LIN {X 0,Y 385.59,Z 292.202,A -85,B 0,C 180,E1 18203.536,E2 18203.536} C_VEL
LIN {X 0,Y 385.578,Z 292.169,A -85,B 0,C 180,E1 18199.701,E2 18199.701} C_VEL
LIN {X 0,Y 385.573,Z 292.168,A -85,B 0,C 180,E1 18195.8,E2 18195.8} C_VEL
LIN {X 0,Y 385.58,Z 292.204,A -85,B 0,C 180,E1 18191.821,E2 18191.821} C_VEL
LIN {X 0,Y 385.579,Z 292.173,A -85,B 0,C 180,E1 18187.75,E2 18187.75} C_VEL
LIN {X 0,Y 385.579,Z 292.168,A -85,B 0,C 180,E1 18183.717,E2 18183.717} C_VEL
LIN {X 0,Y 385.585,Z 292.205,A -85,B 0,C 180,E1 18179.703,E2 18179.703} C_VEL
LIN {X 0,Y 385.583,Z 292.167,A -85,B 0,C 180,E1 18175.687,E2 18175.687} C_VEL
LIN {X 0,Y 385.585,Z 292.173,A -85,B 0,C 180,E1 18171.65,E2 18171.65} C_VEL
LIN {X 0,Y 385.589,Z 292.205,A -85,B 0,C 180,E1 18167.571,E2 18167.571} C_VEL
LIN {X 0,Y 385.589,Z 292.169,A -85,B 0,C 180,E1 18163.582,E2 18163.582} C_VEL
LIN {X 0,Y 385.597,Z 292.203,A -85,B 0,C 180,E1 18159.668,E2 18159.668} C_VEL
LIN {X 0,Y 385.607,Z 292.202,A -85,B 0,C 180,E1 18155.815,E2 18155.815} C_VEL
LIN {X 0,Y 385.613,Z 292.203,A -85,B 0,C 180,E1 18151.831,E2 18151.831} C_VEL
LIN {X 0,Y 385.617,Z 292.201,A -85,B 0,C 180,E1 18147.891,E2 18147.891} C_VEL
LIN {X 0,Y 385.62,Z 292.2,A -85,B 0,C 180,E1 18143.944,E2 18143.944} C_VEL
LIN {X 0,Y 385.628,Z 292.199,A -85,B 0,C 180,E1 18139.894,E2 18139.894} C_VEL
LIN {X 0,Y 385.622,Z 292.201,A -85,B 0,C 180,E1 18135.775,E2 18135.775} C_VEL
LIN {X 0,Y 385.627,Z 292.203,A -85,B 0,C 180,E1 18131.692,E2 18131.692} C_VEL
LIN {X 0,Y 385.625,Z 292.202,A -85,B 0,C 180,E1 18127.726,E2 18127.726} C_VEL
LIN {X 0,Y 385.628,Z 292.234,A -85,B 0,C 180,E1 18123.666,E2 18123.666} C_VEL
LIN {X 0,Y 385.77,Z 293.033,A -85,B 0,C 180,E1 18121.396,E2 18121.396} C_VEL
LIN {X 0,Y 387.406,Z 296.314,A -85,B 0,C 180,E1 18118.016,E2 18118.016} C_VEL
LIN {X 0,Y 389.142,Z 297.888,A -85,B 0,C 180,E1 18114.759,E2 18114.759} C_VEL
LIN {X 0,Y 390.851,Z 298.757,A -85,B 0,C 180,E1 18111.3,E2 18111.3} C_VEL
LIN {X 0,Y 392.259,Z 299.662,A -85,B 0,C 180,E1 18107.964,E2 18107.964} C_VEL
LIN {X 0,Y 393.297,Z 301.626,A -85,B 0,C 180,E1 18104.727,E2 18104.727} C_VEL
LIN {X 0,Y 394.199,Z 303.074,A -85,B 0,C 180,E1 18101.262,E2 18101.262} C_VEL
LIN {X 0,Y 394.882,Z 303.844,A -85,B 0,C 180,E1 18097.712,E2 18097.712} C_VEL
LIN {X 0,Y 395.319,Z 304.24,A -85,B 0,C 180,E1 18094.206,E2 18094.206} C_VEL
LIN {X 0,Y 395.491,Z 304.381,A -85,B 0,C 180,E1 18090.724,E2 18090.724} C_VEL
LIN {X 0,Y 395.407,Z 304.311,A -85,B 0,C 180,E1 18087.101,E2 18087.101} C_VEL
LIN {X 0,Y 395.034,Z 303.985,A -85,B 0,C 180,E1 18083.46,E2 18083.46} C_VEL
LIN {X 0,Y 394.383,Z 303.295,A -85,B 0,C 180,E1 18079.778,E2 18079.778} C_VEL
LIN {X 0,Y 393.61,Z 302.209,A -85,B 0,C 180,E1 18076.485,E2 18076.485} C_VEL
LIN {X 0,Y 392.679,Z 300.302,A -85,B 0,C 180,E1 18073.126,E2 18073.126} C_VEL
LIN {X 0,Y 391.442,Z 298.996,A -85,B 0,C 180,E1 18069.985,E2 18069.985} C_VEL
LIN {X 0,Y 389.81,Z 298.272,A -85,B 0,C 180,E1 18066.574,E2 18066.574} C_VEL
LIN {X 0,Y 387.974,Z 296.947,A -85,B 0,C 180,E1 18063.085,E2 18063.085} C_VEL
LIN {X 0,Y 387.725,Z 296.681,A -85,B 0,C 180,E1 18062.634,E2 18062.634} C_VEL
LIN {X 0,Y 387.23,Z 297.203,A -85,B 0,C 180,E1 18061.86,E2 18061.86} C_VEL
LIN {X 0,Y 385.442,Z 301.535,A -85,B 0,C 180,E1 18059.944,E2 18059.944} C_VEL
LIN {X 0,Y 384.858,Z 301.636,A -85,B 0,C 180,E1 18059.176,E2 18059.176} C_VEL
LIN {X 0,Y 383.634,Z 300.068,A -85,B 0,C 180,E1 18057.174,E2 18057.174} C_VEL
LIN {X 0,Y 381.125,Z 298.816,A -85,B 0,C 180,E1 18053.638,E2 18053.638} C_VEL
LIN {X 0,Y 379.099,Z 296.853,A -85,B 0,C 180,E1 18050.842,E2 18050.842} C_VEL
LIN {X 0,Y 377.788,Z 293.814,A -85,B 0,C 180,E1 18048.373,E2 18048.373} C_VEL
LIN {X 0,Y 377.677,Z 293.211,A -85,B 0,C 180,E1 18046.501,E2 18046.501} C_VEL
LIN {X 0,Y 377.676,Z 293.192,A -85,B 0,C 180,E1 18042.388,E2 18042.388} C_VEL
LIN {X 0,Y 377.672,Z 293.193,A -85,B 0,C 180,E1 18038.407,E2 18038.407} C_VEL
LIN {X 0,Y 377.67,Z 293.192,A -85,B 0,C 180,E1 18034.312,E2 18034.312} C_VEL
LIN {X 0,Y 377.668,Z 293.193,A -85,B 0,C 180,E1 18030.34,E2 18030.34} C_VEL
LIN {X 0,Y 377.662,Z 293.192,A -85,B 0,C 180,E1 18026.409,E2 18026.409} C_VEL
LIN {X 0,Y 377.657,Z 293.194,A -85,B 0,C 180,E1 18022.411,E2 18022.411} C_VEL
LIN {X 0,Y 377.658,Z 293.194,A -85,B 0,C 180,E1 18018.364,E2 18018.364} C_VEL
LIN {X 0,Y 377.651,Z 293.162,A -85,B 0,C 180,E1 18014.254,E2 18014.254} C_VEL
LIN {X 0,Y 377.648,Z 293.151,A -85,B 0,C 180,E1 18010.218,E2 18010.218} C_VEL
LIN {X 0,Y 377.65,Z 293.194,A -85,B 0,C 180,E1 18006.232,E2 18006.232} C_VEL
LIN {X 0,Y 377.645,Z 293.16,A -85,B 0,C 180,E1 18002.124,E2 18002.124} C_VEL
LIN {X 0,Y 377.641,Z 293.155,A -85,B 0,C 180,E1 17998.179,E2 17998.179} C_VEL
LIN {X 0,Y 377.646,Z 293.194,A -85,B 0,C 180,E1 17994.073,E2 17994.073} C_VEL
LIN {X 0,Y 377.638,Z 293.157,A -85,B 0,C 180,E1 17990.031,E2 17990.031} C_VEL
LIN {X 0,Y 377.634,Z 293.159,A -85,B 0,C 180,E1 17986.058,E2 17986.058} C_VEL
LIN {X 0,Y 377.639,Z 293.195,A -85,B 0,C 180,E1 17981.954,E2 17981.954} C_VEL
LIN {X 0,Y 377.633,Z 293.172,A -85,B 0,C 180,E1 17977.916,E2 17977.916} C_VEL
LIN {X 0,Y 377.631,Z 293.159,A -85,B 0,C 180,E1 17973.838,E2 17973.838} C_VEL
LIN {X 0,Y 377.655,Z 293.299,A -85,B 0,C 180,E1 17970.237,E2 17970.237} C_VEL
LIN {X 0,Y 378.612,Z 296.099,A -85,B 0,C 180,E1 17969.269,E2 17969.269} C_VEL
LIN {X 0,Y 383.609,Z 302.624,A -85,B 0,C 180,E1 17967.79,E2 17967.79} C_VEL
LIN {X 0,Y 391.931,Z 314.43,A -85,B 0,C 180,E1 17965.549,E2 17965.549} C_VEL
LIN {X 0,Y 395.837,Z 319.96,A -85,B 0,C 180,E1 17964.571,E2 17964.571} C_VEL
LIN {X 0,Y 403.618,Z 331.65,A -85,B 0,C 180,E1 17962.722,E2 17962.722} C_VEL
LIN {X 0,Y 410.877,Z 343.12,A -85,B 0,C 180,E1 17961.109,E2 17961.109} C_VEL
LIN {X 0,Y 420.09,Z 358.902,A -85,B 0,C 180,E1 17959.184,E2 17959.184} C_VEL
LIN {X 0,Y 426.598,Z 371.081,A -85,B 0,C 180,E1 17957.891,E2 17957.891} C_VEL
LIN {X 0,Y 418.324,Z 587.742,A -85,B 0,C 180,E1 17953.875,E2 17953.875} C_VEL
LIN {X 0,Y 416.849,Z 613.236,A -85,B 0,C 180,E1 17953.319,E2 17953.319} C_VEL
LIN {X 0,Y 415.022,Z 632.082,A -85,B 0,C 180,E1 17952.735,E2 17952.735} C_VEL
LIN {X 0,Y 412.471,Z 653.444,A -85,B 0,C 180,E1 17951.852,E2 17951.852} C_VEL
LIN {X 0,Y 409.295,Z 674.289,A -85,B 0,C 180,E1 17950.71,E2 17950.71} C_VEL
LIN {X 0,Y 406.38,Z 691.177,A -85,B 0,C 180,E1 17949.585,E2 17949.585} C_VEL
LIN {X 0,Y 402.808,Z 710.1,A -85,B 0,C 180,E1 17948.084,E2 17948.084} C_VEL
LIN {X 0,Y 398.872,Z 728.796,A -85,B 0,C 180,E1 17946.268,E2 17946.268} C_VEL
LIN {X 0,Y 395.578,Z 743.764,A -85,B 0,C 180,E1 17944.571,E2 17944.571} C_VEL
LIN {X 0,Y 391.775,Z 760.597,A -85,B 0,C 180,E1 17942.355,E2 17942.355} C_VEL
LIN {X 0,Y 388.258,Z 775.729,A -85,B 0,C 180,E1 17939.972,E2 17939.972} C_VEL
LIN {X 0,Y 385.567,Z 787.594,A -85,B 0,C 180,E1 17937.825,E2 17937.825} C_VEL
LIN {X 0,Y 382.708,Z 800.935,A -85,B 0,C 180,E1 17935.039,E2 17935.039} C_VEL
LIN {X 0,Y 380.326,Z 812.676,A -85,B 0,C 180,E1 17932.082,E2 17932.082} C_VEL
LIN {X 0,Y 378.728,Z 821.683,A -85,B 0,C 180,E1 17929.429,E2 17929.429} C_VEL
LIN {X 0,Y 377.359,Z 830.966,A -85,B 0,C 180,E1 17926.153,E2 17926.153} C_VEL
LIN {X 0,Y 376.588,Z 837.631,A -85,B 0,C 180,E1 17923.199,E2 17923.199} C_VEL
LIN {X 0,Y 376.187,Z 842.608,A -85,B 0,C 180,E1 17920.451,E2 17920.451} C_VEL
LIN {X 0,Y 375.986,Z 846.946,A -85,B 0,C 180,E1 17917.291,E2 17917.291} C_VEL
LIN {X 0,Y 375.927,Z 849.714,A -85,B 0,C 180,E1 17913.965,E2 17913.965} C_VEL
LIN {X 0,Y 375.926,Z 850.752,A -85,B 0,C 180,E1 17911.372,E2 17911.372} C_VEL
LIN {X 0,Y 375.928,Z 850.78,A -85,B 0,C 180,E1 17908.781,E2 17908.781} C_VEL
LIN {X 0,Y 375.927,Z 849.797,A -85,B 0,C 180,E1 17906.188,E2 17906.188} C_VEL
LIN {X 0,Y 375.969,Z 847.379,A -85,B 0,C 180,E1 17903.127,E2 17903.127} C_VEL
LIN {X 0,Y 376.166,Z 842.922,A -85,B 0,C 180,E1 17899.742,E2 17899.742} C_VEL
LIN {X 0,Y 376.558,Z 837.942,A -85,B 0,C 180,E1 17896.957,E2 17896.957} C_VEL
LIN {X 0,Y 377.309,Z 831.337,A -85,B 0,C 180,E1 17894.003,E2 17894.003} C_VEL
LIN {X 0,Y 378.651,Z 822.182,A -85,B 0,C 180,E1 17890.727,E2 17890.727} C_VEL
LIN {X 0,Y 380.22,Z 813.244,A -85,B 0,C 180,E1 17888.074,E2 17888.074} C_VEL
LIN {X 0,Y 382.277,Z 802.862,A -85,B 0,C 180,E1 17885.427,E2 17885.427} C_VEL
LIN {X 0,Y 385.215,Z 789.2,A -85,B 0,C 180,E1 17882.484,E2 17882.484} C_VEL
LIN {X 0,Y 388.052,Z 776.624,A -85,B 0,C 180,E1 17880.18,E2 17880.18} C_VEL
LIN {X 0,Y 391.238,Z 762.786,A -85,B 0,C 180,E1 17877.976,E2 17877.976} C_VEL
LIN {X 0,Y 395.321,Z 744.936,A -85,B 0,C 180,E1 17875.57,E2 17875.57} C_VEL
LIN {X 0,Y 398.708,Z 729.554,A -85,B 0,C 180,E1 17873.812,E2 17873.812} C_VEL
LIN {X 0,Y 402.305,Z 712.451,A -85,B 0,C 180,E1 17872.131,E2 17872.131} C_VEL
LIN {X 0,Y 406.204,Z 692.165,A -85,B 0,C 180,E1 17870.486,E2 17870.486} C_VEL
LIN {X 0,Y 409.103,Z 675.423,A -85,B 0,C 180,E1 17869.359,E2 17869.359} C_VEL
LIN {X 0,Y 411.972,Z 656.79,A -85,B 0,C 180,E1 17868.319,E2 17868.319} C_VEL
LIN {X 0,Y 414.823,Z 634.055,A -85,B 0,C 180,E1 17867.336,E2 17867.336} C_VEL
LIN {X 0,Y 416.669,Z 615.37,A -85,B 0,C 180,E1 17866.74,E2 17866.74} C_VEL
LIN {X 0,Y 418.066,Z 594.306,A -85,B 0,C 180,E1 17866.25,E2 17866.25} C_VEL
LIN {X 0,Y 426.442,Z 375.04,A -85,B 0,C 180,E1 17862.183,E2 17862.183} C_VEL
LIN {X 0,Y 426.491,Z 370.624,A -85,B 0,C 180,E1 17862.082,E2 17862.082} C_VEL
LIN {X 0,Y 416.389,Z 352.336,A -85,B 0,C 180,E1 17860.056,E2 17860.056} C_VEL
LIN {X 0,Y 405.621,Z 334.64,A -85,B 0,C 180,E1 17857.73,E2 17857.73} C_VEL
LIN {X 0,Y 396.092,Z 320.326,A -85,B 0,C 180,E1 17855.492,E2 17855.492} C_VEL
LIN {X 0,Y 392.43,Z 315.132,A -85,B 0,C 180,E1 17854.579,E2 17854.579} C_VEL
LIN {X 0,Y 386.918,Z 307.383,A -85,B 0,C 180,E1 17853.131,E2 17853.131} C_VEL
LIN {X 0,Y 383.245,Z 302.265,A -85,B 0,C 180,E1 17852.111,E2 17852.111} C_VEL
LIN {X 0,Y 378.455,Z 295.814,A -85,B 0,C 180,E1 17850.657,E2 17850.657} C_VEL
LIN {X 0,Y 377.652,Z 293.269,A -85,B 0,C 180,E1 17849.729,E2 17849.729} C_VEL
LIN {X 0,Y 377.637,Z 293.156,A -85,B 0,C 180,E1 17845.735,E2 17845.735} C_VEL
LIN {X 0,Y 377.631,Z 293.166,A -85,B 0,C 180,E1 17841.921,E2 17841.921} C_VEL
LIN {X 0,Y 377.639,Z 293.192,A -85,B 0,C 180,E1 17837.886,E2 17837.886} C_VEL
LIN {X 0,Y 377.635,Z 293.159,A -85,B 0,C 180,E1 17833.786,E2 17833.786} C_VEL
LIN {X 0,Y 377.637,Z 293.153,A -85,B 0,C 180,E1 17829.756,E2 17829.756} C_VEL
LIN {X 0,Y 377.644,Z 293.195,A -85,B 0,C 180,E1 17825.774,E2 17825.774} C_VEL
LIN {X 0,Y 377.641,Z 293.158,A -85,B 0,C 180,E1 17821.669,E2 17821.669} C_VEL
LIN {X 0,Y 377.643,Z 293.157,A -85,B 0,C 180,E1 17817.724,E2 17817.724} C_VEL
LIN {X 0,Y 377.648,Z 293.194,A -85,B 0,C 180,E1 17813.616,E2 17813.616} C_VEL
LIN {X 0,Y 377.647,Z 293.155,A -85,B 0,C 180,E1 17809.474,E2 17809.474} C_VEL
LIN {X 0,Y 377.647,Z 293.157,A -85,B 0,C 180,E1 17805.432,E2 17805.432} C_VEL
LIN {X 0,Y 377.657,Z 293.194,A -85,B 0,C 180,E1 17801.316,E2 17801.316} C_VEL
LIN {X 0,Y 377.659,Z 293.193,A -85,B 0,C 180,E1 17797.261,E2 17797.261} C_VEL
LIN {X 0,Y 377.663,Z 293.192,A -85,B 0,C 180,E1 17793.148,E2 17793.148} C_VEL
LIN {X 0,Y 377.663,Z 293.19,A -85,B 0,C 180,E1 17789.066,E2 17789.066} C_VEL
LIN {X 0,Y 377.664,Z 293.191,A -85,B 0,C 180,E1 17785.12,E2 17785.12} C_VEL
LIN {X 0,Y 377.664,Z 293.19,A -85,B 0,C 180,E1 17781.109,E2 17781.109} C_VEL
LIN {X 0,Y 377.666,Z 293.189,A -85,B 0,C 180,E1 17777.125,E2 17777.125} C_VEL
LIN {X 0,Y 377.671,Z 293.229,A -85,B 0,C 180,E1 17773.056,E2 17773.056} C_VEL
LIN {X 0,Y 377.86,Z 294.198,A -85,B 0,C 180,E1 17771.213,E2 17771.213} C_VEL
LIN {X 0,Y 379.306,Z 297.127,A -85,B 0,C 180,E1 17768.855,E2 17768.855} C_VEL
LIN {X 0,Y 381.485,Z 299.049,A -85,B 0,C 180,E1 17765.916,E2 17765.916} C_VEL
LIN {X 0,Y 384.034,Z 300.4,A -85,B 0,C 180,E1 17762.257,E2 17762.257} C_VEL
LIN {X 0,Y 385.148,Z 302.283,A -85,B 0,C 180,E1 17760.326,E2 17760.326} C_VEL
LIN {X 0,Y 386.727,Z 304.625,A -85,B 0,C 180,E1 17757.4,E2 17757.4} C_VEL
LIN {X 0,Y 388.497,Z 306.031,A -85,B 0,C 180,E1 17754.155,E2 17754.155} C_VEL
LIN {X 0,Y 390.264,Z 306.859,A -85,B 0,C 180,E1 17750.548,E2 17750.548} C_VEL
LIN {X 0,Y 391.49,Z 307.922,A -85,B 0,C 180,E1 17747.386,E2 17747.386} C_VEL
LIN {X 0,Y 392.489,Z 309.904,A -85,B 0,C 180,E1 17744.005,E2 17744.005} C_VEL
LIN {X 0,Y 393.317,Z 311.132,A -85,B 0,C 180,E1 17740.694,E2 17740.694} C_VEL
LIN {X 0,Y 393.988,Z 311.849,A -85,B 0,C 180,E1 17737.29,E2 17737.29} C_VEL
LIN {X 0,Y 394.418,Z 312.249,A -85,B 0,C 180,E1 17733.633,E2 17733.633} C_VEL
LIN {X 0,Y 394.573,Z 312.362,A -85,B 0,C 180,E1 17730,E2 17730} C_VEL
LIN {X 0,Y 394.419,Z 312.25,A -85,B 0,C 180,E1 17726.367,E2 17726.367} C_VEL
LIN {X 0,Y 393.988,Z 311.849,A -85,B 0,C 180,E1 17722.71,E2 17722.71} C_VEL
LIN {X 0,Y 393.294,Z 311.102,A -85,B 0,C 180,E1 17719.157,E2 17719.157} C_VEL
LIN {X 0,Y 392.451,Z 309.82,A -85,B 0,C 180,E1 17715.843,E2 17715.843} C_VEL
LIN {X 0,Y 391.374,Z 307.737,A -85,B 0,C 180,E1 17712.302,E2 17712.302} C_VEL
LIN {X 0,Y 390.013,Z 306.761,A -85,B 0,C 180,E1 17708.967,E2 17708.967} C_VEL
LIN {X 0,Y 388.245,Z 305.89,A -85,B 0,C 180,E1 17705.38,E2 17705.38} C_VEL
LIN {X 0,Y 386.47,Z 304.328,A -85,B 0,C 180,E1 17702.078,E2 17702.078} C_VEL
LIN {X 0,Y 384.882,Z 301.692,A -85,B 0,C 180,E1 17699.219,E2 17699.219} C_VEL
LIN {X 0,Y 384.858,Z 301.636,A -85,B 0,C 180,E1 17699.176,E2 17699.176} C_VEL
LIN {X 0,Y 384.246,Z 301.381,A -85,B 0,C 180,E1 17698.194,E2 17698.194} C_VEL
LIN {X 0,Y 382.956,Z 303.453,A -85,B 0,C 180,E1 17696.736,E2 17696.736} C_VEL
LIN {X 0,Y 381.184,Z 306.655,A -85,B 0,C 180,E1 17694.862,E2 17694.862} C_VEL
LIN {X 0,Y 380.383,Z 306.928,A -85,B 0,C 180,E1 17693.941,E2 17693.941} C_VEL
LIN {X 0,Y 378.223,Z 305,A -85,B 0,C 180,E1 17691.006,E2 17691.006} C_VEL
LIN {X 0,Y 376.839,Z 302.509,A -85,B 0,C 180,E1 17689.011,E2 17689.011} C_VEL
LIN {X 0,Y 375.463,Z 300.938,A -85,B 0,C 180,E1 17687.231,E2 17687.231} C_VEL
LIN {X 0,Y 372.507,Z 299.283,A -85,B 0,C 180,E1 17683.779,E2 17683.779} C_VEL
LIN {X 0,Y 370.823,Z 297.29,A -85,B 0,C 180,E1 17681.758,E2 17681.758} C_VEL
LIN {X 0,Y 369.822,Z 294.627,A -85,B 0,C 180,E1 17679.843,E2 17679.843} C_VEL
LIN {X 0,Y 369.729,Z 294.177,A -85,B 0,C 180,E1 17677.085,E2 17677.085} C_VEL
LIN {X 0,Y 369.725,Z 294.179,A -85,B 0,C 180,E1 17672.927,E2 17672.927} C_VEL
LIN {X 0,Y 369.721,Z 294.18,A -85,B 0,C 180,E1 17668.775,E2 17668.775} C_VEL
LIN {X 0,Y 369.72,Z 294.183,A -85,B 0,C 180,E1 17664.612,E2 17664.612} C_VEL
LIN {X 0,Y 369.718,Z 294.182,A -85,B 0,C 180,E1 17660.583,E2 17660.583} C_VEL
LIN {X 0,Y 369.708,Z 294.145,A -85,B 0,C 180,E1 17656.497,E2 17656.497} C_VEL
LIN {X 0,Y 369.712,Z 294.182,A -85,B 0,C 180,E1 17652.336,E2 17652.336} C_VEL
LIN {X 0,Y 369.71,Z 294.149,A -85,B 0,C 180,E1 17648.192,E2 17648.192} C_VEL
LIN {X 0,Y 369.706,Z 294.139,A -85,B 0,C 180,E1 17644.187,E2 17644.187} C_VEL
LIN {X 0,Y 369.708,Z 294.183,A -85,B 0,C 180,E1 17640.155,E2 17640.155} C_VEL
LIN {X 0,Y 369.701,Z 294.144,A -85,B 0,C 180,E1 17636.123,E2 17636.123} C_VEL
LIN {X 0,Y 369.7,Z 294.145,A -85,B 0,C 180,E1 17632.072,E2 17632.072} C_VEL
LIN {X 0,Y 369.704,Z 294.184,A -85,B 0,C 180,E1 17627.981,E2 17627.981} C_VEL
LIN {X 0,Y 369.697,Z 294.148,A -85,B 0,C 180,E1 17623.987,E2 17623.987} C_VEL
LIN {X 0,Y 369.694,Z 294.144,A -85,B 0,C 180,E1 17619.911,E2 17619.911} C_VEL
LIN {X 0,Y 369.695,Z 294.165,A -85,B 0,C 180,E1 17615.897,E2 17615.897} C_VEL
LIN {X 0,Y 369.719,Z 294.354,A -85,B 0,C 180,E1 17612.017,E2 17612.017} C_VEL
LIN {X 0,Y 370.014,Z 295.612,A -85,B 0,C 180,E1 17611.58,E2 17611.58} C_VEL
LIN {X 0,Y 371.953,Z 298.759,A -85,B 0,C 180,E1 17610.886,E2 17610.886} C_VEL
LIN {X 0,Y 374.407,Z 301.301,A -85,B 0,C 180,E1 17610.129,E2 17610.129} C_VEL
LIN {X 0,Y 381.676,Z 310.922,A -85,B 0,C 180,E1 17607.962,E2 17607.962} C_VEL
LIN {X 0,Y 388.476,Z 320.636,A -85,B 0,C 180,E1 17606.092,E2 17606.092} C_VEL
LIN {X 0,Y 395.873,Z 331.318,A -85,B 0,C 180,E1 17604.218,E2 17604.218} C_VEL
LIN {X 0,Y 404.594,Z 345.229,A -85,B 0,C 180,E1 17602.158,E2 17602.158} C_VEL
LIN {X 0,Y 413.34,Z 359.909,A -85,B 0,C 180,E1 17600.244,E2 17600.244} C_VEL
LIN {X 0,Y 421.1,Z 374.389,A -85,B 0,C 180,E1 17598.635,E2 17598.635} C_VEL
LIN {X 0,Y 412.376,Z 592.617,A -85,B 0,C 180,E1 17594.552,E2 17594.552} C_VEL
LIN {X 0,Y 410.888,Z 614.663,A -85,B 0,C 180,E1 17594.041,E2 17594.041} C_VEL
LIN {X 0,Y 408.974,Z 633.378,A -85,B 0,C 180,E1 17593.445,E2 17593.445} C_VEL
LIN {X 0,Y 406.172,Z 655.22,A -85,B 0,C 180,E1 17592.509,E2 17592.509} C_VEL
LIN {X 0,Y 403.179,Z 674.037,A -85,B 0,C 180,E1 17591.462,E2 17591.462} C_VEL
LIN {X 0,Y 400.137,Z 690.924,A -85,B 0,C 180,E1 17590.328,E2 17590.328} C_VEL
LIN {X 0,Y 396.328,Z 710.208,A -85,B 0,C 180,E1 17588.781,E2 17588.781} C_VEL
LIN {X 0,Y 392.272,Z 728.541,A -85,B 0,C 180,E1 17586.979,E2 17586.979} C_VEL
LIN {X 0,Y 388.813,Z 743.507,A -85,B 0,C 180,E1 17585.261,E2 17585.261} C_VEL
LIN {X 0,Y 384.767,Z 760.538,A -85,B 0,C 180,E1 17582.983,E2 17582.983} C_VEL
LIN {X 0,Y 381.096,Z 775.471,A -85,B 0,C 180,E1 17580.595,E2 17580.595} C_VEL
LIN {X 0,Y 378.108,Z 787.963,A -85,B 0,C 180,E1 17578.288,E2 17578.288} C_VEL
LIN {X 0,Y 374.904,Z 801.963,A -85,B 0,C 180,E1 17575.259,E2 17575.259} C_VEL
LIN {X 0,Y 372.668,Z 812.419,A -85,B 0,C 180,E1 17572.56,E2 17572.56} C_VEL
LIN {X 0,Y 370.945,Z 821.498,A -85,B 0,C 180,E1 17569.83,E2 17569.83} C_VEL
LIN {X 0,Y 369.425,Z 831.082,A -85,B 0,C 180,E1 17566.348,E2 17566.348} C_VEL
LIN {X 0,Y 368.644,Z 837.378,A -85,B 0,C 180,E1 17563.488,E2 17563.488} C_VEL
LIN {X 0,Y 368.226,Z 842.167,A -85,B 0,C 180,E1 17560.798,E2 17560.798} C_VEL
LIN {X 0,Y 368.011,Z 846.061,A -85,B 0,C 180,E1 17557.964,E2 17557.964} C_VEL
LIN {X 0,Y 367.934,Z 849.216,A -85,B 0,C 180,E1 17554.52,E2 17554.52} C_VEL
LIN {X 0,Y 367.927,Z 850.476,A -85,B 0,C 180,E1 17551.557,E2 17551.557} C_VEL
LIN {X 0,Y 367.933,Z 850.559,A -85,B 0,C 180,E1 17548.91,E2 17548.91} C_VEL
LIN {X 0,Y 367.928,Z 849.63,A -85,B 0,C 180,E1 17546.261,E2 17546.261} C_VEL
LIN {X 0,Y 367.957,Z 847.544,A -85,B 0,C 180,E1 17543.447,E2 17543.447} C_VEL
LIN {X 0,Y 368.143,Z 843.424,A -85,B 0,C 180,E1 17539.99,E2 17539.99} C_VEL
LIN {X 0,Y 368.574,Z 838.092,A -85,B 0,C 180,E1 17536.876,E2 17536.876} C_VEL
LIN {X 0,Y 369.267,Z 832.195,A -85,B 0,C 180,E1 17534.129,E2 17534.129} C_VEL
LIN {X 0,Y 370.555,Z 823.897,A -85,B 0,C 180,E1 17530.945,E2 17530.945} C_VEL
LIN {X 0,Y 372.441,Z 813.555,A -85,B 0,C 180,E1 17527.758,E2 17527.758} C_VEL
LIN {X 0,Y 374.471,Z 803.843,A -85,B 0,C 180,E1 17525.205,E2 17525.205} C_VEL
LIN {X 0,Y 377.519,Z 790.549,A -85,B 0,C 180,E1 17522.217,E2 17522.217} C_VEL
LIN {X 0,Y 380.669,Z 777.261,A -85,B 0,C 180,E1 17519.716,E2 17519.716} C_VEL
LIN {X 0,Y 383.874,Z 764.023,A -85,B 0,C 180,E1 17517.551,E2 17517.551} C_VEL
LIN {X 0,Y 387.838,Z 747.825,A -85,B 0,C 180,E1 17515.269,E2 17515.269} C_VEL
LIN {X 0,Y 391.775,Z 730.758,A -85,B 0,C 180,E1 17513.261,E2 17513.261} C_VEL
LIN {X 0,Y 395.189,Z 715.282,A -85,B 0,C 180,E1 17511.695,E2 17511.695} C_VEL
LIN {X 0,Y 399.242,Z 695.804,A -85,B 0,C 180,E1 17510.027,E2 17510.027} C_VEL
LIN {X 0,Y 402.784,Z 676.304,A -85,B 0,C 180,E1 17508.678,E2 17508.678} C_VEL
LIN {X 0,Y 405.552,Z 659.177,A -85,B 0,C 180,E1 17507.698,E2 17507.698} C_VEL
LIN {X 0,Y 408.491,Z 638.046,A -85,B 0,C 180,E1 17506.726,E2 17506.726} C_VEL
LIN {X 0,Y 410.707,Z 616.797,A -85,B 0,C 180,E1 17506.019,E2 17506.019} C_VEL
LIN {X 0,Y 412.091,Z 597.739,A -85,B 0,C 180,E1 17505.557,E2 17505.557} C_VEL
LIN {X 0,Y 420.835,Z 380.823,A -85,B 0,C 180,E1 17501.486,E2 17501.486} C_VEL
LIN {X 0,Y 420.998,Z 373.973,A -85,B 0,C 180,E1 17501.339,E2 17501.339} C_VEL
LIN {X 0,Y 411.068,Z 356.061,A -85,B 0,C 180,E1 17499.273,E2 17499.273} C_VEL
LIN {X 0,Y 401.693,Z 340.462,A -85,B 0,C 180,E1 17497.173,E2 17497.173} C_VEL
LIN {X 0,Y 392.696,Z 326.713,A -85,B 0,C 180,E1 17494.996,E2 17494.996} C_VEL
LIN {X 0,Y 384.265,Z 314.547,A -85,B 0,C 180,E1 17492.766,E2 17492.766} C_VEL
LIN {X 0,Y 380.162,Z 308.907,A -85,B 0,C 180,E1 17491.604,E2 17491.604} C_VEL
LIN {X 0,Y 373.306,Z 299.933,A -85,B 0,C 180,E1 17489.526,E2 17489.526} C_VEL
LIN {X 0,Y 370.672,Z 297.093,A -85,B 0,C 180,E1 17488.694,E2 17488.694} C_VEL
LIN {X 0,Y 369.77,Z 294.672,A -85,B 0,C 180,E1 17488.179,E2 17488.179} C_VEL
LIN {X 0,Y 369.735,Z 294.154,A -85,B 0,C 180,E1 17487.168,E2 17487.168} C_VEL
LIN {X 0,Y 369.74,Z 294.174,A -85,B 0,C 180,E1 17482.918,E2 17482.918} C_VEL
LIN {X 0,Y 369.728,Z 294.157,A -85,B 0,C 180,E1 17478.773,E2 17478.773} C_VEL
LIN {X 0,Y 369.732,Z 294.132,A -85,B 0,C 180,E1 17474.726,E2 17474.726} C_VEL
LIN {X 0,Y 369.726,Z 294.15,A -85,B 0,C 180,E1 17470.597,E2 17470.597} C_VEL
LIN {X 0,Y 369.732,Z 294.173,A -85,B 0,C 180,E1 17466.522,E2 17466.522} C_VEL
LIN {X 0,Y 369.728,Z 294.133,A -85,B 0,C 180,E1 17462.48,E2 17462.48} C_VEL
LIN {X 0,Y 369.735,Z 294.156,A -85,B 0,C 180,E1 17458.45,E2 17458.45} C_VEL
LIN {X 0,Y 369.729,Z 294.169,A -85,B 0,C 180,E1 17454.257,E2 17454.257} C_VEL
LIN {X 0,Y 369.733,Z 294.133,A -85,B 0,C 180,E1 17450.348,E2 17450.348} C_VEL
LIN {X 0,Y 369.741,Z 294.156,A -85,B 0,C 180,E1 17446.233,E2 17446.233} C_VEL
LIN {X 0,Y 369.739,Z 294.172,A -85,B 0,C 180,E1 17442.15,E2 17442.15} C_VEL
LIN {X 0,Y 369.741,Z 294.18,A -85,B 0,C 180,E1 17438.051,E2 17438.051} C_VEL
LIN {X 0,Y 369.74,Z 294.181,A -85,B 0,C 180,E1 17434.018,E2 17434.018} C_VEL
LIN {X 0,Y 369.742,Z 294.178,A -85,B 0,C 180,E1 17429.919,E2 17429.919} C_VEL
LIN {X 0,Y 369.734,Z 294.179,A -85,B 0,C 180,E1 17425.772,E2 17425.772} C_VEL
LIN {X 0,Y 369.738,Z 294.201,A -85,B 0,C 180,E1 17421.647,E2 17421.647} C_VEL
LIN {X 0,Y 369.862,Z 294.842,A -85,B 0,C 180,E1 17419.909,E2 17419.909} C_VEL
LIN {X 0,Y 371.757,Z 298.582,A -85,B 0,C 180,E1 17417.121,E2 17417.121} C_VEL
LIN {X 0,Y 374.183,Z 300.379,A -85,B 0,C 180,E1 17414.265,E2 17414.265} C_VEL
LIN {X 0,Y 376.356,Z 301.679,A -85,B 0,C 180,E1 17411.71,E2 17411.71} C_VEL
LIN {X 0,Y 378.228,Z 305.006,A -85,B 0,C 180,E1 17408.987,E2 17408.987} C_VEL
LIN {X 0,Y 380.465,Z 306.978,A -85,B 0,C 180,E1 17405.961,E2 17405.961} C_VEL
LIN {X 0,Y 382.977,Z 308.302,A -85,B 0,C 180,E1 17402.357,E2 17402.357} C_VEL
LIN {X 0,Y 384.056,Z 310.137,A -85,B 0,C 180,E1 17400.489,E2 17400.489} C_VEL
LIN {X 0,Y 385.705,Z 312.542,A -85,B 0,C 180,E1 17397.478,E2 17397.478} C_VEL
LIN {X 0,Y 387.493,Z 313.958,A -85,B 0,C 180,E1 17394.221,E2 17394.221} C_VEL
LIN {X 0,Y 389.259,Z 314.79,A -85,B 0,C 180,E1 17390.603,E2 17390.603} C_VEL
LIN {X 0,Y 390.491,Z 315.868,A -85,B 0,C 180,E1 17387.432,E2 17387.432} C_VEL
LIN {X 0,Y 391.523,Z 317.886,A -85,B 0,C 180,E1 17383.968,E2 17383.968} C_VEL
LIN {X 0,Y 392.392,Z 319.136,A -85,B 0,C 180,E1 17380.423,E2 17380.423} C_VEL
LIN {X 0,Y 393.048,Z 319.827,A -85,B 0,C 180,E1 17376.867,E2 17376.867} C_VEL
LIN {X 0,Y 393.449,Z 320.185,A -85,B 0,C 180,E1 17373.351,E2 17373.351} C_VEL
LIN {X 0,Y 393.585,Z 320.295,A -85,B 0,C 180,E1 17369.854,E2 17369.854} C_VEL
LIN {X 0,Y 393.43,Z 320.185,A -85,B 0,C 180,E1 17366.211,E2 17366.211} C_VEL
LIN {X 0,Y 392.995,Z 319.784,A -85,B 0,C 180,E1 17362.545,E2 17362.545} C_VEL
LIN {X 0,Y 392.275,Z 318.996,A -85,B 0,C 180,E1 17358.906,E2 17358.906} C_VEL
LIN {X 0,Y 391.395,Z 317.62,A -85,B 0,C 180,E1 17355.502,E2 17355.502} C_VEL
LIN {X 0,Y 390.324,Z 315.594,A -85,B 0,C 180,E1 17352.098,E2 17352.098} C_VEL
LIN {X 0,Y 389.006,Z 314.69,A -85,B 0,C 180,E1 17348.909,E2 17348.909} C_VEL
LIN {X 0,Y 387.244,Z 313.825,A -85,B 0,C 180,E1 17345.348,E2 17345.348} C_VEL
LIN {X 0,Y 385.45,Z 312.243,A -85,B 0,C 180,E1 17341.998,E2 17341.998} C_VEL
LIN {X 0,Y 383.836,Z 309.638,A -85,B 0,C 180,E1 17339.126,E2 17339.126} C_VEL
LIN {X 0,Y 382.712,Z 308.08,A -85,B 0,C 180,E1 17337.263,E2 17337.263} C_VEL
LIN {X 0,Y 380.383,Z 306.928,A -85,B 0,C 180,E1 17333.941,E2 17333.941} C_VEL
LIN {X 0,Y 379.269,Z 307.369,A -85,B 0,C 180,E1 17332.617,E2 17332.617} C_VEL
LIN {X 0,Y 376.641,Z 310.471,A -85,B 0,C 180,E1 17329.908,E2 17329.908} C_VEL
LIN {X 0,Y 375.679,Z 310.213,A -85,B 0,C 180,E1 17328.75,E2 17328.75} C_VEL
LIN {X 0,Y 375.627,Z 310.114,A -85,B 0,C 180,E1 17328.668,E2 17328.668} C_VEL
LIN {X 0,Y 374.161,Z 308.759,A -85,B 0,C 180,E1 17326.837,E2 17326.837} C_VEL
LIN {X 0,Y 371.34,Z 307.107,A -85,B 0,C 180,E1 17323.574,E2 17323.574} C_VEL
LIN {X 0,Y 369.619,Z 305.035,A -85,B 0,C 180,E1 17321.51,E2 17321.51} C_VEL
LIN {X 0,Y 367.97,Z 302.23,A -85,B 0,C 180,E1 17319.481,E2 17319.481} C_VEL
LIN {X 0,Y 364.61,Z 300.309,A -85,B 0,C 180,E1 17315.933,E2 17315.933} C_VEL
LIN {X 0,Y 362.806,Z 298.156,A -85,B 0,C 180,E1 17313.952,E2 17313.952} C_VEL
LIN {X 0,Y 361.891,Z 295.785,A -85,B 0,C 180,E1 17312.411,E2 17312.411} C_VEL
LIN {X 0,Y 361.789,Z 295.189,A -85,B 0,C 180,E1 17310.933,E2 17310.933} C_VEL
LIN {X 0,Y 361.784,Z 295.17,A -85,B 0,C 180,E1 17306.774,E2 17306.774} C_VEL
LIN {X 0,Y 361.778,Z 295.171,A -85,B 0,C 180,E1 17302.591,E2 17302.591} C_VEL
LIN {X 0,Y 361.782,Z 295.172,A -85,B 0,C 180,E1 17298.365,E2 17298.365} C_VEL
LIN {X 0,Y 361.774,Z 295.136,A -85,B 0,C 180,E1 17294.239,E2 17294.239} C_VEL
LIN {X 0,Y 361.771,Z 295.125,A -85,B 0,C 180,E1 17290.188,E2 17290.188} C_VEL
LIN {X 0,Y 361.773,Z 295.171,A -85,B 0,C 180,E1 17286.188,E2 17286.188} C_VEL
LIN {X 0,Y 361.769,Z 295.135,A -85,B 0,C 180,E1 17282.059,E2 17282.059} C_VEL
LIN {X 0,Y 361.764,Z 295.128,A -85,B 0,C 180,E1 17278.099,E2 17278.099} C_VEL
LIN {X 0,Y 361.77,Z 295.172,A -85,B 0,C 180,E1 17273.971,E2 17273.971} C_VEL
LIN {X 0,Y 361.766,Z 295.134,A -85,B 0,C 180,E1 17269.812,E2 17269.812} C_VEL
LIN {X 0,Y 361.763,Z 295.129,A -85,B 0,C 180,E1 17265.76,E2 17265.76} C_VEL
LIN {X 0,Y 361.769,Z 295.161,A -85,B 0,C 180,E1 17261.635,E2 17261.635} C_VEL
LIN {X 0,Y 361.763,Z 295.153,A -85,B 0,C 180,E1 17257.579,E2 17257.579} C_VEL
LIN {X 0,Y 361.79,Z 295.334,A -85,B 0,C 180,E1 17254.351,E2 17254.351} C_VEL
LIN {X 0,Y 362.081,Z 296.61,A -85,B 0,C 180,E1 17253.912,E2 17253.912} C_VEL
LIN {X 0,Y 363.839,Z 299.574,A -85,B 0,C 180,E1 17253.212,E2 17253.212} C_VEL
LIN {X 0,Y 367.026,Z 302.146,A -85,B 0,C 180,E1 17252.147,E2 17252.147} C_VEL
LIN {X 0,Y 369.482,Z 305.9,A -85,B 0,C 180,E1 17251.293,E2 17251.293} C_VEL
LIN {X 0,Y 372.117,Z 308.742,A -85,B 0,C 180,E1 17250.459,E2 17250.459} C_VEL
LIN {X 0,Y 378.943,Z 318.053,A -85,B 0,C 180,E1 17248.371,E2 17248.371} C_VEL
LIN {X 0,Y 384.938,Z 326.656,A -85,B 0,C 180,E1 17246.677,E2 17246.677} C_VEL
LIN {X 0,Y 392.894,Z 338.453,A -85,B 0,C 180,E1 17244.601,E2 17244.601} C_VEL
LIN {X 0,Y 400.99,Z 351.543,A -85,B 0,C 180,E1 17242.638,E2 17242.638} C_VEL
LIN {X 0,Y 409.433,Z 365.971,A -85,B 0,C 180,E1 17240.737,E2 17240.737} C_VEL
LIN {X 0,Y 415.673,Z 377.757,A -85,B 0,C 180,E1 17239.398,E2 17239.398} C_VEL
LIN {X 0,Y 406.479,Z 596.25,A -85,B 0,C 180,E1 17235.265,E2 17235.265} C_VEL
LIN {X 0,Y 404.997,Z 616.09,A -85,B 0,C 180,E1 17234.784,E2 17234.784} C_VEL
LIN {X 0,Y 402.771,Z 636.723,A -85,B 0,C 180,E1 17234.101,E2 17234.101} C_VEL
LIN {X 0,Y 399.716,Z 658.238,A -85,B 0,C 180,E1 17233.119,E2 17233.119} C_VEL
LIN {X 0,Y 396.931,Z 674.919,A -85,B 0,C 180,E1 17232.167,E2 17232.167} C_VEL
LIN {X 0,Y 393.792,Z 691.56,A -85,B 0,C 180,E1 17231.03,E2 17231.03} C_VEL
LIN {X 0,Y 389.515,Z 711.942,A -85,B 0,C 180,E1 17229.347,E2 17229.347} C_VEL
LIN {X 0,Y 385.574,Z 728.974,A -85,B 0,C 180,E1 17227.638,E2 17227.638} C_VEL
LIN {X 0,Y 381.814,Z 744.486,A -85,B 0,C 180,E1 17225.822,E2 17225.822} C_VEL
LIN {X 0,Y 377.183,Z 762.77,A -85,B 0,C 180,E1 17223.279,E2 17223.279} C_VEL
LIN {X 0,Y 373.754,Z 776.108,A -85,B 0,C 180,E1 17221.084,E2 17221.084} C_VEL
LIN {X 0,Y 370.586,Z 788.685,A -85,B 0,C 180,E1 17218.701,E2 17218.701} C_VEL
LIN {X 0,Y 367.262,Z 802.347,A -85,B 0,C 180,E1 17215.649,E2 17215.649} C_VEL
LIN {X 0,Y 364.912,Z 812.73,A -85,B 0,C 180,E1 17212.897,E2 17212.897} C_VEL
LIN {X 0,Y 363.023,Z 822.168,A -85,B 0,C 180,E1 17209.969,E2 17209.969} C_VEL
LIN {X 0,Y 361.495,Z 831.198,A -85,B 0,C 180,E1 17206.552,E2 17206.552} C_VEL
LIN {X 0,Y 360.672,Z 837.435,A -85,B 0,C 180,E1 17203.629,E2 17203.629} C_VEL
LIN {X 0,Y 360.214,Z 842.443,A -85,B 0,C 180,E1 17200.702,E2 17200.702} C_VEL
LIN {X 0,Y 359.987,Z 846.879,A -85,B 0,C 180,E1 17197.18,E2 17197.18} C_VEL
LIN {X 0,Y 359.932,Z 849.299,A -85,B 0,C 180,E1 17193.982,E2 17193.982} C_VEL
LIN {X 0,Y 359.935,Z 850.283,A -85,B 0,C 180,E1 17191.273,E2 17191.273} C_VEL
LIN {X 0,Y 359.932,Z 850.255,A -85,B 0,C 180,E1 17188.567,E2 17188.567} C_VEL
LIN {X 0,Y 359.937,Z 849.133,A -85,B 0,C 180,E1 17185.699,E2 17185.699} C_VEL
LIN {X 0,Y 360.004,Z 846.198,A -85,B 0,C 180,E1 17182.179,E2 17182.179} C_VEL
LIN {X 0,Y 360.234,Z 842.166,A -85,B 0,C 180,E1 17179.121,E2 17179.121} C_VEL
LIN {X 0,Y 360.673,Z 837.435,A -85,B 0,C 180,E1 17176.371,E2 17176.371} C_VEL
LIN {X 0,Y 361.495,Z 831.198,A -85,B 0,C 180,E1 17173.448,E2 17173.448} C_VEL
LIN {X 0,Y 363.113,Z 821.669,A -85,B 0,C 180,E1 17169.868,E2 17169.868} C_VEL
LIN {X 0,Y 364.912,Z 812.73,A -85,B 0,C 180,E1 17167.103,E2 17167.103} C_VEL
LIN {X 0,Y 367.262,Z 802.347,A -85,B 0,C 180,E1 17164.351,E2 17164.351} C_VEL
LIN {X 0,Y 370.647,Z 788.434,A -85,B 0,C 180,E1 17161.249,E2 17161.249} C_VEL
LIN {X 0,Y 373.843,Z 775.757,A -85,B 0,C 180,E1 17158.854,E2 17158.854} C_VEL
LIN {X 0,Y 377.485,Z 761.657,A -85,B 0,C 180,E1 17156.548,E2 17156.548} C_VEL
LIN {X 0,Y 381.96,Z 743.869,A -85,B 0,C 180,E1 17154.102,E2 17154.102} C_VEL
LIN {X 0,Y 385.574,Z 728.974,A -85,B 0,C 180,E1 17152.362,E2 17152.362} C_VEL
LIN {X 0,Y 389.515,Z 711.942,A -85,B 0,C 180,E1 17150.653,E2 17150.653} C_VEL
LIN {X 0,Y 393.792,Z 691.56,A -85,B 0,C 180,E1 17148.97,E2 17148.97} C_VEL
LIN {X 0,Y 396.931,Z 674.919,A -85,B 0,C 180,E1 17147.833,E2 17147.833} C_VEL
LIN {X 0,Y 399.828,Z 657.543,A -85,B 0,C 180,E1 17146.844,E2 17146.844} C_VEL
LIN {X 0,Y 402.977,Z 634.809,A -85,B 0,C 180,E1 17145.829,E2 17145.829} C_VEL
LIN {X 0,Y 405.065,Z 615.328,A -85,B 0,C 180,E1 17145.194,E2 17145.194} C_VEL
LIN {X 0,Y 406.529,Z 595.195,A -85,B 0,C 180,E1 17144.714,E2 17144.714} C_VEL
LIN {X 0,Y 415.681,Z 377.529,A -85,B 0,C 180,E1 17140.597,E2 17140.597} C_VEL
LIN {X 0,Y 405.044,Z 358.186,A -85,B 0,C 180,E1 17138.287,E2 17138.287} C_VEL
LIN {X 0,Y 396.702,Z 344.58,A -85,B 0,C 180,E1 17136.343,E2 17136.343} C_VEL
LIN {X 0,Y 389.206,Z 332.919,A -85,B 0,C 180,E1 17134.459,E2 17134.459} C_VEL
LIN {X 0,Y 381.15,Z 321.134,A -85,B 0,C 180,E1 17132.265,E2 17132.265} C_VEL
LIN {X 0,Y 377.02,Z 315.427,A -85,B 0,C 180,E1 17131.061,E2 17131.061} C_VEL
LIN {X 0,Y 370.789,Z 307.102,A -85,B 0,C 180,E1 17129.117,E2 17129.117} C_VEL
LIN {X 0,Y 367.907,Z 303.828,A -85,B 0,C 180,E1 17128.177,E2 17128.177} C_VEL
LIN {X 0,Y 366.614,Z 301.611,A -85,B 0,C 180,E1 17127.71,E2 17127.71} C_VEL
LIN {X 0,Y 363.338,Z 298.987,A -85,B 0,C 180,E1 17126.607,E2 17126.607} C_VEL
LIN {X 0,Y 361.861,Z 295.767,A -85,B 0,C 180,E1 17125.885,E2 17125.885} C_VEL
LIN {X 0,Y 361.788,Z 295.13,A -85,B 0,C 180,E1 17125.189,E2 17125.189} C_VEL
LIN {X 0,Y 361.797,Z 295.124,A -85,B 0,C 180,E1 17121.055,E2 17121.055} C_VEL
LIN {X 0,Y 361.796,Z 295.144,A -85,B 0,C 180,E1 17116.869,E2 17116.869} C_VEL
LIN {X 0,Y 361.797,Z 295.151,A -85,B 0,C 180,E1 17112.773,E2 17112.773} C_VEL
LIN {X 0,Y 361.788,Z 295.121,A -85,B 0,C 180,E1 17108.583,E2 17108.583} C_VEL
LIN {X 0,Y 361.793,Z 295.141,A -85,B 0,C 180,E1 17104.597,E2 17104.597} C_VEL
LIN {X 0,Y 361.798,Z 295.156,A -85,B 0,C 180,E1 17100.475,E2 17100.475} C_VEL
LIN {X 0,Y 361.787,Z 295.12,A -85,B 0,C 180,E1 17096.356,E2 17096.356} C_VEL
LIN {X 0,Y 361.79,Z 295.143,A -85,B 0,C 180,E1 17092.217,E2 17092.217} C_VEL
LIN {X 0,Y 361.784,Z 295.16,A -85,B 0,C 180,E1 17088.037,E2 17088.037} C_VEL
LIN {X 0,Y 361.783,Z 295.126,A -85,B 0,C 180,E1 17083.956,E2 17083.956} C_VEL
LIN {X 0,Y 361.792,Z 295.169,A -85,B 0,C 180,E1 17079.959,E2 17079.959} C_VEL
LIN {X 0,Y 361.793,Z 295.169,A -85,B 0,C 180,E1 17075.857,E2 17075.857} C_VEL
LIN {X 0,Y 361.795,Z 295.17,A -85,B 0,C 180,E1 17071.798,E2 17071.798} C_VEL
LIN {X 0,Y 361.848,Z 295.478,A -85,B 0,C 180,E1 17067.959,E2 17067.959} C_VEL
LIN {X 0,Y 362.338,Z 297.201,A -85,B 0,C 180,E1 17066.598,E2 17066.598} C_VEL
LIN {X 0,Y 363.8,Z 299.548,A -85,B 0,C 180,E1 17064.942,E2 17064.942} C_VEL
LIN {X 0,Y 366.237,Z 301.362,A -85,B 0,C 180,E1 17062.345,E2 17062.345} C_VEL
LIN {X 0,Y 368.376,Z 302.645,A -85,B 0,C 180,E1 17060.065,E2 17060.065} C_VEL
LIN {X 0,Y 370.578,Z 306.36,A -85,B 0,C 180,E1 17057.373,E2 17057.373} C_VEL
LIN {X 0,Y 372.978,Z 308.219,A -85,B 0,C 180,E1 17054.514,E2 17054.514} C_VEL
LIN {X 0,Y 375.147,Z 309.443,A -85,B 0,C 180,E1 17051.961,E2 17051.961} C_VEL
LIN {X 0,Y 377.153,Z 312.885,A -85,B 0,C 180,E1 17049.119,E2 17049.119} C_VEL
LIN {X 0,Y 379.294,Z 314.816,A -85,B 0,C 180,E1 17046.19,E2 17046.19} C_VEL
LIN {X 0,Y 381.87,Z 316.16,A -85,B 0,C 180,E1 17042.531,E2 17042.531} C_VEL
LIN {X 0,Y 382.893,Z 317.825,A -85,B 0,C 180,E1 17040.782,E2 17040.782} C_VEL
LIN {X 0,Y 384.599,Z 320.357,A -85,B 0,C 180,E1 17037.732,E2 17037.732} C_VEL
LIN {X 0,Y 386.486,Z 321.885,A -85,B 0,C 180,E1 17034.288,E2 17034.288} C_VEL
LIN {X 0,Y 388.255,Z 322.721,A -85,B 0,C 180,E1 17030.659,E2 17030.659} C_VEL
LIN {X 0,Y 389.492,Z 323.812,A -85,B 0,C 180,E1 17027.478,E2 17027.478} C_VEL
LIN {X 0,Y 390.539,Z 325.833,A -85,B 0,C 180,E1 17023.996,E2 17023.996} C_VEL
LIN {X 0,Y 391.415,Z 327.077,A -85,B 0,C 180,E1 17020.433,E2 17020.433} C_VEL
LIN {X 0,Y 392.072,Z 327.766,A -85,B 0,C 180,E1 17016.884,E2 17016.884} C_VEL
LIN {X 0,Y 392.476,Z 328.126,A -85,B 0,C 180,E1 17013.359,E2 17013.359} C_VEL
LIN {X 0,Y 392.596,Z 328.228,A -85,B 0,C 180,E1 17009.708,E2 17009.708} C_VEL
LIN {X 0,Y 392.443,Z 328.105,A -85,B 0,C 180,E1 17006.056,E2 17006.056} C_VEL
LIN {X 0,Y 391.972,Z 327.697,A -85,B 0,C 180,E1 17002.378,E2 17002.378} C_VEL
LIN {X 0,Y 391.277,Z 326.919,A -85,B 0,C 180,E1 16998.802,E2 16998.802} C_VEL
LIN {X 0,Y 390.345,Z 325.436,A -85,B 0,C 180,E1 16995.159,E2 16995.159} C_VEL
LIN {X 0,Y 389.271,Z 323.449,A -85,B 0,C 180,E1 16991.871,E2 16991.871} C_VEL
LIN {X 0,Y 387.841,Z 322.547,A -85,B 0,C 180,E1 16988.527,E2 16988.527} C_VEL
LIN {X 0,Y 385.983,Z 321.582,A -85,B 0,C 180,E1 16984.861,E2 16984.861} C_VEL
LIN {X 0,Y 384.214,Z 319.951,A -85,B 0,C 180,E1 16981.561,E2 16981.561} C_VEL
LIN {X 0,Y 382.696,Z 317.35,A -85,B 0,C 180,E1 16978.849,E2 16978.849} C_VEL
LIN {X 0,Y 381.535,Z 315.884,A -85,B 0,C 180,E1 16976.97,E2 16976.97} C_VEL
LIN {X 0,Y 378.929,Z 314.57,A -85,B 0,C 180,E1 16973.335,E2 16973.335} C_VEL
LIN {X 0,Y 376.877,Z 312.497,A -85,B 0,C 180,E1 16970.453,E2 16970.453} C_VEL
LIN {X 0,Y 375.627,Z 310.114,A -85,B 0,C 180,E1 16968.668,E2 16968.668} C_VEL
LIN {X 0,Y 375.065,Z 310.178,A -85,B 0,C 180,E1 16967.996,E2 16967.996} C_VEL
LIN {X 0,Y 373.775,Z 312.7,A -85,B 0,C 180,E1 16966.921,E2 16966.921} C_VEL
LIN {X 0,Y 372.282,Z 315.704,A -85,B 0,C 180,E1 16965.726,E2 16965.726} C_VEL
LIN {X 0,Y 371.712,Z 316.023,A -85,B 0,C 180,E1 16965.151,E2 16965.151} C_VEL
LIN {X 0,Y 369.034,Z 313.753,A -85,B 0,C 180,E1 16962.007,E2 16962.007} C_VEL
LIN {X 0,Y 366.796,Z 310.054,A -85,B 0,C 180,E1 16959.273,E2 16959.273} C_VEL
LIN {X 0,Y 363.545,Z 308.235,A -85,B 0,C 180,E1 16955.86,E2 16955.86} C_VEL
LIN {X 0,Y 361.622,Z 305.999,A -85,B 0,C 180,E1 16953.762,E2 16953.762} C_VEL
LIN {X 0,Y 360.116,Z 303.325,A -85,B 0,C 180,E1 16952.026,E2 16952.026} C_VEL
LIN {X 0,Y 356.549,Z 301.218,A -85,B 0,C 180,E1 16948.472,E2 16948.472} C_VEL
LIN {X 0,Y 354.641,Z 298.775,A -85,B 0,C 180,E1 16946.633,E2 16946.633} C_VEL
LIN {X 0,Y 353.967,Z 296.757,A -85,B 0,C 180,E1 16945.606,E2 16945.606} C_VEL
LIN {X 0,Y 353.852,Z 296.16,A -85,B 0,C 180,E1 16944.187,E2 16944.187} C_VEL
LIN {X 0,Y 353.848,Z 296.158,A -85,B 0,C 180,E1 16940.165,E2 16940.165} C_VEL
LIN {X 0,Y 353.84,Z 296.114,A -85,B 0,C 180,E1 16936.077,E2 16936.077} C_VEL
LIN {X 0,Y 353.841,Z 296.15,A -85,B 0,C 180,E1 16932.07,E2 16932.07} C_VEL
LIN {X 0,Y 353.84,Z 296.127,A -85,B 0,C 180,E1 16927.959,E2 16927.959} C_VEL
LIN {X 0,Y 353.837,Z 296.11,A -85,B 0,C 180,E1 16923.889,E2 16923.889} C_VEL
LIN {X 0,Y 353.839,Z 296.154,A -85,B 0,C 180,E1 16919.838,E2 16919.838} C_VEL
LIN {X 0,Y 353.842,Z 296.124,A -85,B 0,C 180,E1 16915.624,E2 16915.624} C_VEL
LIN {X 0,Y 353.841,Z 296.111,A -85,B 0,C 180,E1 16911.551,E2 16911.551} C_VEL
LIN {X 0,Y 353.847,Z 296.148,A -85,B 0,C 180,E1 16907.433,E2 16907.433} C_VEL
LIN {X 0,Y 353.848,Z 296.131,A -85,B 0,C 180,E1 16903.31,E2 16903.31} C_VEL
LIN {X 0,Y 353.852,Z 296.114,A -85,B 0,C 180,E1 16899.143,E2 16899.143} C_VEL
LIN {X 0,Y 353.9,Z 296.413,A -85,B 0,C 180,E1 16897.053,E2 16897.053} C_VEL
LIN {X 0,Y 354.281,Z 297.964,A -85,B 0,C 180,E1 16896.511,E2 16896.511} C_VEL
LIN {X 0,Y 356.097,Z 300.801,A -85,B 0,C 180,E1 16895.711,E2 16895.711} C_VEL
LIN {X 0,Y 359.287,Z 303.112,A -85,B 0,C 180,E1 16894.513,E2 16894.513} C_VEL
LIN {X 0,Y 361.477,Z 306.719,A -85,B 0,C 180,E1 16893.644,E2 16893.644} C_VEL
LIN {X 0,Y 364.59,Z 309.503,A -85,B 0,C 180,E1 16892.566,E2 16892.566} C_VEL
LIN {X 0,Y 367.46,Z 313.489,A -85,B 0,C 180,E1 16891.564,E2 16891.564} C_VEL
LIN {X 0,Y 370.38,Z 316.888,A -85,B 0,C 180,E1 16890.617,E2 16890.617} C_VEL
LIN {X 0,Y 376.457,Z 325.495,A -85,B 0,C 180,E1 16888.719,E2 16888.719} C_VEL
LIN {X 0,Y 381.675,Z 333.044,A -85,B 0,C 180,E1 16887.206,E2 16887.206} C_VEL
LIN {X 0,Y 389.687,Z 345.169,A -85,B 0,C 180,E1 16885.053,E2 16885.053} C_VEL
LIN {X 0,Y 398.659,Z 359.83,A -85,B 0,C 180,E1 16882.834,E2 16882.834} C_VEL
LIN {X 0,Y 407.8,Z 376.232,A -85,B 0,C 180,E1 16880.737,E2 16880.737} C_VEL
LIN {X 0,Y 410.313,Z 381.312,A -85,B 0,C 180,E1 16880.178,E2 16880.178} C_VEL
LIN {X 0,Y 400.762,Z 597.629,A -85,B 0,C 180,E1 16876.044,E2 16876.044} C_VEL
LIN {X 0,Y 399.217,Z 617.06,A -85,B 0,C 180,E1 16875.562,E2 16875.562} C_VEL
LIN {X 0,Y 396.759,Z 638.606,A -85,B 0,C 180,E1 16874.827,E2 16874.827} C_VEL
LIN {X 0,Y 393.734,Z 658.675,A -85,B 0,C 180,E1 16873.887,E2 16873.887} C_VEL
LIN {X 0,Y 390.744,Z 675.8,A -85,B 0,C 180,E1 16872.893,E2 16872.893} C_VEL
LIN {X 0,Y 386.956,Z 694.985,A -85,B 0,C 180,E1 16871.547,E2 16871.547} C_VEL
LIN {X 0,Y 382.719,Z 713.752,A -85,B 0,C 180,E1 16869.924,E2 16869.924} C_VEL
LIN {X 0,Y 378.931,Z 729.408,A -85,B 0,C 180,E1 16868.321,E2 16868.321} C_VEL
LIN {X 0,Y 374.853,Z 745.463,A -85,B 0,C 180,E1 16866.403,E2 16866.403} C_VEL
LIN {X 0,Y 370.162,Z 763.011,A -85,B 0,C 180,E1 16863.902,E2 16863.902} C_VEL
LIN {X 0,Y 366.566,Z 776.273,A -85,B 0,C 180,E1 16861.677,E2 16861.677} C_VEL
LIN {X 0,Y 362.929,Z 790.034,A -85,B 0,C 180,E1 16859.003,E2 16859.003} C_VEL
LIN {X 0,Y 359.638,Z 802.73,A -85,B 0,C 180,E1 16856.056,E2 16856.056} C_VEL
LIN {X 0,Y 357.264,Z 812.618,A -85,B 0,C 180,E1 16853.371,E2 16853.371} C_VEL
LIN {X 0,Y 355.183,Z 822.41,A -85,B 0,C 180,E1 16850.258,E2 16850.258} C_VEL
LIN {X 0,Y 353.567,Z 831.314,A -85,B 0,C 180,E1 16846.765,E2 16846.765} C_VEL
LIN {X 0,Y 352.703,Z 837.491,A -85,B 0,C 180,E1 16843.776,E2 16843.776} C_VEL
LIN {X 0,Y 352.205,Z 842.669,A -85,B 0,C 180,E1 16840.633,E2 16840.633} C_VEL
LIN {X 0,Y 351.979,Z 846.906,A -85,B 0,C 180,E1 16837.016,E2 16837.016} C_VEL
LIN {X 0,Y 351.936,Z 849.05,A -85,B 0,C 180,E1 16834.073,E2 16834.073} C_VEL
LIN {X 0,Y 351.938,Z 850.035,A -85,B 0,C 180,E1 16831.302,E2 16831.302} C_VEL
LIN {X 0,Y 351.936,Z 850.007,A -85,B 0,C 180,E1 16828.535,E2 16828.535} C_VEL
LIN {X 0,Y 351.939,Z 848.884,A -85,B 0,C 180,E1 16825.601,E2 16825.601} C_VEL
LIN {X 0,Y 352.013,Z 845.948,A -85,B 0,C 180,E1 16822,E2 16822} C_VEL
LIN {X 0,Y 352.261,Z 841.914,A -85,B 0,C 180,E1 16818.872,E2 16818.872} C_VEL
LIN {X 0,Y 352.739,Z 837.181,A -85,B 0,C 180,E1 16816.059,E2 16816.059} C_VEL
LIN {X 0,Y 353.694,Z 830.572,A -85,B 0,C 180,E1 16812.903,E2 16812.903} C_VEL
LIN {X 0,Y 355.376,Z 821.413,A -85,B 0,C 180,E1 16809.41,E2 16809.41} C_VEL
LIN {X 0,Y 357.296,Z 812.473,A -85,B 0,C 180,E1 16806.587,E2 16806.587} C_VEL
LIN {X 0,Y 359.801,Z 802.089,A -85,B 0,C 180,E1 16803.779,E2 16803.779} C_VEL
LIN {X 0,Y 363.33,Z 788.427,A -85,B 0,C 180,E1 16800.671,E2 16800.671} C_VEL
LIN {X 0,Y 366.678,Z 775.851,A -85,B 0,C 180,E1 16798.247,E2 16798.247} C_VEL
LIN {X 0,Y 370.395,Z 762.186,A -85,B 0,C 180,E1 16795.968,E2 16795.968} C_VEL
LIN {X 0,Y 375.159,Z 744.229,A -85,B 0,C 180,E1 16793.441,E2 16793.441} C_VEL
LIN {X 0,Y 379.12,Z 728.65,A -85,B 0,C 180,E1 16791.596,E2 16791.596} C_VEL
LIN {X 0,Y 383.328,Z 711.288,A -85,B 0,C 180,E1 16789.84,E2 16789.84} C_VEL
LIN {X 0,Y 387.639,Z 691.529,A -85,B 0,C 180,E1 16788.196,E2 16788.196} C_VEL
LIN {X 0,Y 390.975,Z 674.553,A -85,B 0,C 180,E1 16787.028,E2 16787.028} C_VEL
LIN {X 0,Y 394.022,Z 656.943,A -85,B 0,C 180,E1 16786.02,E2 16786.02} C_VEL
LIN {X 0,Y 397.314,Z 633.841,A -85,B 0,C 180,E1 16784.992,E2 16784.992} C_VEL
LIN {X 0,Y 399.43,Z 614.773,A -85,B 0,C 180,E1 16784.373,E2 16784.373} C_VEL
LIN {X 0,Y 400.973,Z 594.007,A -85,B 0,C 180,E1 16783.878,E2 16783.878} C_VEL
LIN {X 0,Y 410.328,Z 380.935,A -85,B 0,C 180,E1 16779.815,E2 16779.815} C_VEL
LIN {X 0,Y 400.685,Z 363.315,A -85,B 0,C 180,E1 16777.643,E2 16777.643} C_VEL
LIN {X 0,Y 391.314,Z 347.699,A -85,B 0,C 180,E1 16775.362,E2 16775.362} C_VEL
LIN {X 0,Y 382.98,Z 334.991,A -85,B 0,C 180,E1 16773.158,E2 16773.158} C_VEL
LIN {X 0,Y 377.715,Z 327.267,A -85,B 0,C 180,E1 16771.654,E2 16771.654} C_VEL
LIN {X 0,Y 373.869,Z 321.862,A -85,B 0,C 180,E1 16770.495,E2 16770.495} C_VEL
LIN {X 0,Y 368.336,Z 314.295,A -85,B 0,C 180,E1 16768.716,E2 16768.716} C_VEL
LIN {X 0,Y 365.174,Z 310.557,A -85,B 0,C 180,E1 16767.652,E2 16767.652} C_VEL
LIN {X 0,Y 363.974,Z 308.789,A -85,B 0,C 180,E1 16767.218,E2 16767.218} C_VEL
LIN {X 0,Y 360.791,Z 305.869,A -85,B 0,C 180,E1 16766.1,E2 16766.1} C_VEL
LIN {X 0,Y 358.858,Z 302.596,A -85,B 0,C 180,E1 16765.321,E2 16765.321} C_VEL
LIN {X 0,Y 355.637,Z 300.303,A -85,B 0,C 180,E1 16764.102,E2 16764.102} C_VEL
LIN {X 0,Y 354.021,Z 297.082,A -85,B 0,C 180,E1 16763.291,E2 16763.291} C_VEL
LIN {X 0,Y 353.846,Z 296.194,A -85,B 0,C 180,E1 16762.688,E2 16762.688} C_VEL
LIN {X 0,Y 353.841,Z 296.135,A -85,B 0,C 180,E1 16758.621,E2 16758.621} C_VEL
LIN {X 0,Y 353.842,Z 296.109,A -85,B 0,C 180,E1 16754.566,E2 16754.566} C_VEL
LIN {X 0,Y 353.836,Z 296.122,A -85,B 0,C 180,E1 16750.419,E2 16750.419} C_VEL
LIN {X 0,Y 353.842,Z 296.155,A -85,B 0,C 180,E1 16746.327,E2 16746.327} C_VEL
LIN {X 0,Y 353.832,Z 296.112,A -85,B 0,C 180,E1 16742.105,E2 16742.105} C_VEL
LIN {X 0,Y 353.834,Z 296.123,A -85,B 0,C 180,E1 16738.057,E2 16738.057} C_VEL
LIN {X 0,Y 353.835,Z 296.157,A -85,B 0,C 180,E1 16733.836,E2 16733.836} C_VEL
LIN {X 0,Y 353.829,Z 296.115,A -85,B 0,C 180,E1 16729.581,E2 16729.581} C_VEL
LIN {X 0,Y 353.831,Z 296.119,A -85,B 0,C 180,E1 16725.434,E2 16725.434} C_VEL
LIN {X 0,Y 353.845,Z 296.159,A -85,B 0,C 180,E1 16721.188,E2 16721.188} C_VEL
LIN {X 0,Y 353.848,Z 296.159,A -85,B 0,C 180,E1 16717.049,E2 16717.049} C_VEL
LIN {X 0,Y 353.927,Z 296.569,A -85,B 0,C 180,E1 16714.57,E2 16714.57} C_VEL
LIN {X 0,Y 354.677,Z 298.846,A -85,B 0,C 180,E1 16713.332,E2 16713.332} C_VEL
LIN {X 0,Y 356.549,Z 301.218,A -85,B 0,C 180,E1 16711.528,E2 16711.528} C_VEL
LIN {X 0,Y 360.375,Z 303.615,A -85,B 0,C 180,E1 16707.718,E2 16707.718} C_VEL
LIN {X 0,Y 362.592,Z 307.318,A -85,B 0,C 180,E1 16705.194,E2 16705.194} C_VEL
LIN {X 0,Y 365.049,Z 309.216,A -85,B 0,C 180,E1 16702.551,E2 16702.551} C_VEL
LIN {X 0,Y 367.238,Z 310.515,A -85,B 0,C 180,E1 16700.222,E2 16700.222} C_VEL
LIN {X 0,Y 369.372,Z 314.134,A -85,B 0,C 180,E1 16697.622,E2 16697.622} C_VEL
LIN {X 0,Y 371.959,Z 316.151,A -85,B 0,C 180,E1 16694.553,E2 16694.553} C_VEL
LIN {X 0,Y 374.11,Z 317.397,A -85,B 0,C 180,E1 16692.013,E2 16692.013} C_VEL
LIN {X 0,Y 376.079,Z 320.764,A -85,B 0,C 180,E1 16689.252,E2 16689.252} C_VEL
LIN {X 0,Y 378.248,Z 322.73,A -85,B 0,C 180,E1 16686.271,E2 16686.271} C_VEL
LIN {X 0,Y 380.738,Z 323.994,A -85,B 0,C 180,E1 16682.749,E2 16682.749} C_VEL
LIN {X 0,Y 381.749,Z 325.531,A -85,B 0,C 180,E1 16681.062,E2 16681.062} C_VEL
LIN {X 0,Y 383.4,Z 328.075,A -85,B 0,C 180,E1 16678.165,E2 16678.165} C_VEL
LIN {X 0,Y 385.254,Z 329.704,A -85,B 0,C 180,E1 16674.698,E2 16674.698} C_VEL
LIN {X 0,Y 387.08,Z 330.587,A -85,B 0,C 180,E1 16671.041,E2 16671.041} C_VEL
LIN {X 0,Y 388.387,Z 331.545,A -85,B 0,C 180,E1 16667.839,E2 16667.839} C_VEL
LIN {X 0,Y 389.495,Z 333.649,A -85,B 0,C 180,E1 16664.266,E2 16664.266} C_VEL
LIN {X 0,Y 390.381,Z 334.944,A -85,B 0,C 180,E1 16660.776,E2 16660.776} C_VEL
LIN {X 0,Y 391.073,Z 335.674,A -85,B 0,C 180,E1 16657.197,E2 16657.197} C_VEL
LIN {X 0,Y 391.48,Z 336.068,A -85,B 0,C 180,E1 16653.661,E2 16653.661} C_VEL
LIN {X 0,Y 391.648,Z 336.183,A -85,B 0,C 180,E1 16650,E2 16650} C_VEL
LIN {X 0,Y 391.48,Z 336.069,A -85,B 0,C 180,E1 16646.339,E2 16646.339} C_VEL
LIN {X 0,Y 391.063,Z 335.669,A -85,B 0,C 180,E1 16642.656,E2 16642.656} C_VEL
LIN {X 0,Y 390.35,Z 334.914,A -85,B 0,C 180,E1 16639.074,E2 16639.074} C_VEL
LIN {X 0,Y 389.461,Z 333.568,A -85,B 0,C 180,E1 16635.58,E2 16635.58} C_VEL
LIN {X 0,Y 388.387,Z 331.545,A -85,B 0,C 180,E1 16632.161,E2 16632.161} C_VEL
LIN {X 0,Y 387.081,Z 330.587,A -85,B 0,C 180,E1 16628.959,E2 16628.959} C_VEL
LIN {X 0,Y 385.243,Z 329.696,A -85,B 0,C 180,E1 16625.283,E2 16625.283} C_VEL
LIN {X 0,Y 383.393,Z 328.066,A -85,B 0,C 180,E1 16621.821,E2 16621.821} C_VEL
LIN {X 0,Y 381.702,Z 325.412,A -85,B 0,C 180,E1 16618.847,E2 16618.847} C_VEL
LIN {X 0,Y 380.695,Z 323.958,A -85,B 0,C 180,E1 16617.187,E2 16617.187} C_VEL
LIN {X 0,Y 378.058,Z 322.602,A -85,B 0,C 180,E1 16613.484,E2 16613.484} C_VEL
LIN {X 0,Y 375.901,Z 320.522,A -85,B 0,C 180,E1 16610.477,E2 16610.477} C_VEL
LIN {X 0,Y 373.78,Z 317.056,A -85,B 0,C 180,E1 16607.586,E2 16607.586} C_VEL
LIN {X 0,Y 371.712,Z 316.023,A -85,B 0,C 180,E1 16605.151,E2 16605.151} C_VEL
LIN {X 0,Y 370.932,Z 316.641,A -85,B 0,C 180,E1 16604.35,E2 16604.35} C_VEL
LIN {X 0,Y 368.496,Z 321.159,A -85,B 0,C 180,E1 16602.373,E2 16602.373} C_VEL
LIN {X 0,Y 367.769,Z 321.394,A -85,B 0,C 180,E1 16601.689,E2 16601.689} C_VEL
LIN {X 0,Y 367.672,Z 321.278,A -85,B 0,C 180,E1 16601.576,E2 16601.576} C_VEL
LIN {X 0,Y 365.714,Z 317.95,A -85,B 0,C 180,E1 16599.165,E2 16599.165} C_VEL
LIN {X 0,Y 362.481,Z 316.161,A -85,B 0,C 180,E1 16595.787,E2 16595.787} C_VEL
LIN {X 0,Y 360.467,Z 313.883,A -85,B 0,C 180,E1 16593.598,E2 16593.598} C_VEL
LIN {X 0,Y 358.867,Z 311.093,A -85,B 0,C 180,E1 16591.775,E2 16591.775} C_VEL
LIN {X 0,Y 355.271,Z 308.976,A -85,B 0,C 180,E1 16588.217,E2 16588.217} C_VEL
LIN {X 0,Y 353.339,Z 306.533,A -85,B 0,C 180,E1 16586.377,E2 16586.377} C_VEL
LIN {X 0,Y 352.061,Z 304.247,A -85,B 0,C 180,E1 16585.214,E2 16585.214} C_VEL
LIN {X 0,Y 348.541,Z 302.151,A -85,B 0,C 180,E1 16582.696,E2 16582.696} C_VEL
LIN {X 0,Y 346.694,Z 299.689,A -85,B 0,C 180,E1 16581.397,E2 16581.397} C_VEL
LIN {X 0,Y 345.985,Z 297.673,A -85,B 0,C 180,E1 16580.561,E2 16580.561} C_VEL
LIN {X 0,Y 345.93,Z 297.146,A -85,B 0,C 180,E1 16579.414,E2 16579.414} C_VEL
LIN {X 0,Y 345.912,Z 297.099,A -85,B 0,C 180,E1 16575.116,E2 16575.116} C_VEL
LIN {X 0,Y 345.907,Z 297.109,A -85,B 0,C 180,E1 16570.998,E2 16570.998} C_VEL
LIN {X 0,Y 345.904,Z 297.146,A -85,B 0,C 180,E1 16566.806,E2 16566.806} C_VEL
LIN {X 0,Y 345.892,Z 297.1,A -85,B 0,C 180,E1 16562.651,E2 16562.651} C_VEL
LIN {X 0,Y 345.889,Z 297.108,A -85,B 0,C 180,E1 16558.509,E2 16558.509} C_VEL
LIN {X 0,Y 345.89,Z 297.151,A -85,B 0,C 180,E1 16554.193,E2 16554.193} C_VEL
LIN {X 0,Y 345.883,Z 297.106,A -85,B 0,C 180,E1 16550.012,E2 16550.012} C_VEL
LIN {X 0,Y 345.88,Z 297.106,A -85,B 0,C 180,E1 16545.947,E2 16545.947} C_VEL
LIN {X 0,Y 345.886,Z 297.14,A -85,B 0,C 180,E1 16541.808,E2 16541.808} C_VEL
LIN {X 0,Y 345.932,Z 297.459,A -85,B 0,C 180,E1 16540.235,E2 16540.235} C_VEL
LIN {X 0,Y 346.393,Z 299.08,A -85,B 0,C 180,E1 16539.615,E2 16539.615} C_VEL
LIN {X 0,Y 348.499,Z 302.084,A -85,B 0,C 180,E1 16538.543,E2 16538.543} C_VEL
LIN {X 0,Y 351.587,Z 304.178,A -85,B 0,C 180,E1 16537.203,E2 16537.203} C_VEL
LIN {X 0,Y 353.584,Z 307.665,A -85,B 0,C 180,E1 16536.281,E2 16536.281} C_VEL
LIN {X 0,Y 357.007,Z 310.563,A -85,B 0,C 180,E1 16534.938,E2 16534.938} C_VEL
LIN {X 0,Y 359.678,Z 314.45,A -85,B 0,C 180,E1 16533.88,E2 16533.88} C_VEL
LIN {X 0,Y 362.182,Z 316.784,A -85,B 0,C 180,E1 16532.991,E2 16532.991} C_VEL
LIN {X 0,Y 365.448,Z 321.062,A -85,B 0,C 180,E1 16531.839,E2 16531.839} C_VEL
LIN {X 0,Y 369.162,Z 325.965,A -85,B 0,C 180,E1 16530.6,E2 16530.6} C_VEL
LIN {X 0,Y 377.196,Z 337.319,A -85,B 0,C 180,E1 16528.119,E2 16528.119} C_VEL
LIN {X 0,Y 387.304,Z 353.142,A -85,B 0,C 180,E1 16525.303,E2 16525.303} C_VEL
LIN {X 0,Y 395.732,Z 367.325,A -85,B 0,C 180,E1 16523.171,E2 16523.171} C_VEL
LIN {X 0,Y 404.238,Z 382.886,A -85,B 0,C 180,E1 16521.17,E2 16521.17} C_VEL
LIN {X 0,Y 405.032,Z 384.819,A -85,B 0,C 180,E1 16520.978,E2 16520.978} C_VEL
LIN {X 0,Y 395.133,Z 598.806,A -85,B 0,C 180,E1 16516.851,E2 16516.851} C_VEL
LIN {X 0,Y 393.472,Z 618.487,A -85,B 0,C 180,E1 16516.349,E2 16516.349} C_VEL
LIN {X 0,Y 390.587,Z 641.571,A -85,B 0,C 180,E1 16515.519,E2 16515.519} C_VEL
LIN {X 0,Y 387.717,Z 659.744,A -85,B 0,C 180,E1 16514.645,E2 16514.645} C_VEL
LIN {X 0,Y 384.623,Z 676.681,A -85,B 0,C 180,E1 16513.644,E2 16513.644} C_VEL
LIN {X 0,Y 380.405,Z 696.919,A -85,B 0,C 180,E1 16512.186,E2 16512.186} C_VEL
LIN {X 0,Y 376.032,Z 715.291,A -85,B 0,C 180,E1 16510.549,E2 16510.549} C_VEL
LIN {X 0,Y 371.992,Z 731.218,A -85,B 0,C 180,E1 16508.873,E2 16508.873} C_VEL
LIN {X 0,Y 367.132,Z 749.316,A -85,B 0,C 180,E1 16506.613,E2 16506.613} C_VEL
LIN {X 0,Y 362.898,Z 764.248,A -85,B 0,C 180,E1 16504.389,E2 16504.389} C_VEL
LIN {X 0,Y 359.158,Z 777.384,A -85,B 0,C 180,E1 16502.121,E2 16502.121} C_VEL
LIN {X 0,Y 354.848,Z 792.736,A -85,B 0,C 180,E1 16498.988,E2 16498.988} C_VEL
LIN {X 0,Y 351.863,Z 803.755,A -85,B 0,C 180,E1 16496.313,E2 16496.313} C_VEL
LIN {X 0,Y 349.308,Z 813.919,A -85,B 0,C 180,E1 16493.445,E2 16493.445} C_VEL
LIN {X 0,Y 346.871,Z 824.865,A -85,B 0,C 180,E1 16489.709,E2 16489.709} C_VEL
LIN {X 0,Y 345.545,Z 832.033,A -85,B 0,C 180,E1 16486.711,E2 16486.711} C_VEL
LIN {X 0,Y 344.663,Z 838.169,A -85,B 0,C 180,E1 16483.59,E2 16483.59} C_VEL
LIN {X 0,Y 344.131,Z 843.751,A -85,B 0,C 180,E1 16479.87,E2 16479.87} C_VEL
LIN {X 0,Y 343.97,Z 846.933,A -85,B 0,C 180,E1 16476.845,E2 16476.845} C_VEL
LIN {X 0,Y 343.938,Z 848.884,A -85,B 0,C 180,E1 16474.001,E2 16474.001} C_VEL
LIN {X 0,Y 343.943,Z 849.814,A -85,B 0,C 180,E1 16471.166,E2 16471.166} C_VEL
LIN {X 0,Y 343.938,Z 849.731,A -85,B 0,C 180,E1 16468.334,E2 16468.334} C_VEL
LIN {X 0,Y 343.943,Z 848.385,A -85,B 0,C 180,E1 16464.997,E2 16464.997} C_VEL
LIN {X 0,Y 344.039,Z 845.309,A -85,B 0,C 180,E1 16461.477,E2 16461.477} C_VEL
LIN {X 0,Y 344.311,Z 841.41,A -85,B 0,C 180,E1 16458.442,E2 16458.442} C_VEL
LIN {X 0,Y 344.903,Z 836.306,A -85,B 0,C 180,E1 16455.392,E2 16455.392} C_VEL
LIN {X 0,Y 346.135,Z 828.767,A -85,B 0,C 180,E1 16451.822,E2 16451.822} C_VEL
LIN {X 0,Y 347.868,Z 820.158,A -85,B 0,C 180,E1 16448.591,E2 16448.591} C_VEL
LIN {X 0,Y 350.019,Z 810.976,A -85,B 0,C 180,E1 16445.678,E2 16445.678} C_VEL
LIN {X 0,Y 353.288,Z 798.49,A -85,B 0,C 180,E1 16442.346,E2 16442.346} C_VEL
LIN {X 0,Y 356.555,Z 786.563,A -85,B 0,C 180,E1 16439.686,E2 16439.686} C_VEL
LIN {X 0,Y 360.097,Z 774.09,A -85,B 0,C 180,E1 16437.28,E2 16437.28} C_VEL
LIN {X 0,Y 364.659,Z 758.176,A -85,B 0,C 180,E1 16434.653,E2 16434.653} C_VEL
LIN {X 0,Y 369.07,Z 742.124,A -85,B 0,C 180,E1 16432.444,E2 16432.444} C_VEL
LIN {X 0,Y 373.149,Z 726.781,A -85,B 0,C 180,E1 16430.633,E2 16430.633} C_VEL
LIN {X 0,Y 378.045,Z 707.155,A -85,B 0,C 180,E1 16428.688,E2 16428.688} C_VEL
LIN {X 0,Y 382.043,Z 689.178,A -85,B 0,C 180,E1 16427.224,E2 16427.224} C_VEL
LIN {X 0,Y 385.503,Z 672.075,A -85,B 0,C 180,E1 16426.063,E2 16426.063} C_VEL
LIN {X 0,Y 389.307,Z 650.102,A -85,B 0,C 180,E1 16424.86,E2 16424.86} C_VEL
LIN {X 0,Y 392.058,Z 630.388,A -85,B 0,C 180,E1 16424.043,E2 16424.043} C_VEL
LIN {X 0,Y 394.209,Z 611.009,A -85,B 0,C 180,E1 16423.44,E2 16423.44} C_VEL
LIN {X 0,Y 395.992,Z 581.933,A -85,B 0,C 180,E1 16422.806,E2 16422.806} C_VEL
LIN {X 0,Y 405.044,Z 384.365,A -85,B 0,C 180,E1 16419.011,E2 16419.011} C_VEL
LIN {X 0,Y 396.119,Z 367.996,A -85,B 0,C 180,E1 16416.923,E2 16416.923} C_VEL
LIN {X 0,Y 387.552,Z 353.522,A -85,B 0,C 180,E1 16414.762,E2 16414.762} C_VEL
LIN {X 0,Y 379.608,Z 341.214,A -85,B 0,C 180,E1 16412.591,E2 16412.591} C_VEL
LIN {X 0,Y 374.782,Z 333.992,A -85,B 0,C 180,E1 16411.169,E2 16411.169} C_VEL
LIN {X 0,Y 370.451,Z 327.868,A -85,B 0,C 180,E1 16409.821,E2 16409.821} C_VEL
LIN {X 0,Y 365.881,Z 321.464,A -85,B 0,C 180,E1 16408.303,E2 16408.303} C_VEL
LIN {X 0,Y 362.471,Z 317.285,A -85,B 0,C 180,E1 16407.118,E2 16407.118} C_VEL
LIN {X 0,Y 361.368,Z 315.91,A -85,B 0,C 180,E1 16406.719,E2 16406.719} C_VEL
LIN {X 0,Y 358.087,Z 312.473,A -85,B 0,C 180,E1 16405.512,E2 16405.512} C_VEL
LIN {X 0,Y 356.538,Z 310,A -85,B 0,C 180,E1 16404.876,E2 16404.876} C_VEL
LIN {X 0,Y 353.318,Z 307.336,A -85,B 0,C 180,E1 16403.605,E2 16403.605} C_VEL
LIN {X 0,Y 351.339,Z 303.791,A -85,B 0,C 180,E1 16402.682,E2 16402.682} C_VEL
LIN {X 0,Y 348.006,Z 301.581,A -85,B 0,C 180,E1 16401.224,E2 16401.224} C_VEL
LIN {X 0,Y 346.133,Z 298.341,A -85,B 0,C 180,E1 16400.185,E2 16400.185} C_VEL
LIN {X 0,Y 345.904,Z 297.175,A -85,B 0,C 180,E1 16399.415,E2 16399.415} C_VEL
LIN {X 0,Y 345.912,Z 297.094,A -85,B 0,C 180,E1 16395.116,E2 16395.116} C_VEL
LIN {X 0,Y 345.916,Z 297.115,A -85,B 0,C 180,E1 16390.829,E2 16390.829} C_VEL
LIN {X 0,Y 345.922,Z 297.13,A -85,B 0,C 180,E1 16386.639,E2 16386.639} C_VEL
LIN {X 0,Y 345.902,Z 297.097,A -85,B 0,C 180,E1 16382.319,E2 16382.319} C_VEL
LIN {X 0,Y 345.9,Z 297.112,A -85,B 0,C 180,E1 16378.178,E2 16378.178} C_VEL
LIN {X 0,Y 345.897,Z 297.143,A -85,B 0,C 180,E1 16373.904,E2 16373.904} C_VEL
LIN {X 0,Y 345.891,Z 297.101,A -85,B 0,C 180,E1 16369.676,E2 16369.676} C_VEL
LIN {X 0,Y 345.892,Z 297.106,A -85,B 0,C 180,E1 16365.434,E2 16365.434} C_VEL
LIN {X 0,Y 345.908,Z 297.148,A -85,B 0,C 180,E1 16361.111,E2 16361.111} C_VEL
LIN {X 0,Y 345.962,Z 297.543,A -85,B 0,C 180,E1 16359.531,E2 16359.531} C_VEL
LIN {X 0,Y 346.639,Z 299.581,A -85,B 0,C 180,E1 16358.644,E2 16358.644} C_VEL
LIN {X 0,Y 348.427,Z 302.049,A -85,B 0,C 180,E1 16357.385,E2 16357.385} C_VEL
LIN {X 0,Y 351.859,Z 304.084,A -85,B 0,C 180,E1 16354.95,E2 16354.95} C_VEL
LIN {X 0,Y 353.058,Z 305.939,A -85,B 0,C 180,E1 16353.913,E2 16353.913} C_VEL
LIN {X 0,Y 354.75,Z 308.432,A -85,B 0,C 180,E1 16352.287,E2 16352.287} C_VEL
LIN {X 0,Y 357.522,Z 310.421,A -85,B 0,C 180,E1 16349.59,E2 16349.59} C_VEL
LIN {X 0,Y 359.206,Z 311.469,A -85,B 0,C 180,E1 16347.883,E2 16347.883} C_VEL
LIN {X 0,Y 361.376,Z 315.084,A -85,B 0,C 180,E1 16345.445,E2 16345.445} C_VEL
LIN {X 0,Y 363.994,Z 317.133,A -85,B 0,C 180,E1 16342.622,E2 16342.622} C_VEL
LIN {X 0,Y 366.026,Z 318.263,A -85,B 0,C 180,E1 16340.471,E2 16340.471} C_VEL
LIN {X 0,Y 368.167,Z 321.919,A -85,B 0,C 180,E1 16337.85,E2 16337.85} C_VEL
LIN {X 0,Y 370.828,Z 324.025,A -85,B 0,C 180,E1 16334.725,E2 16334.725} C_VEL
LIN {X 0,Y 373.072,Z 325.354,A -85,B 0,C 180,E1 16332.066,E2 16332.066} C_VEL
LIN {X 0,Y 374.869,Z 328.478,A -85,B 0,C 180,E1 16329.572,E2 16329.572} C_VEL
LIN {X 0,Y 377.06,Z 330.547,A -85,B 0,C 180,E1 16326.537,E2 16326.537} C_VEL
LIN {X 0,Y 379.687,Z 331.896,A -85,B 0,C 180,E1 16322.851,E2 16322.851} C_VEL
LIN {X 0,Y 380.706,Z 333.481,A -85,B 0,C 180,E1 16321.156,E2 16321.156} C_VEL
LIN {X 0,Y 382.391,Z 336.007,A -85,B 0,C 180,E1 16318.216,E2 16318.216} C_VEL
LIN {X 0,Y 384.242,Z 337.632,A -85,B 0,C 180,E1 16314.749,E2 16314.749} C_VEL
LIN {X 0,Y 386.075,Z 338.516,A -85,B 0,C 180,E1 16311.099,E2 16311.099} C_VEL
LIN {X 0,Y 387.392,Z 339.484,A -85,B 0,C 180,E1 16307.886,E2 16307.886} C_VEL
LIN {X 0,Y 388.511,Z 341.592,A -85,B 0,C 180,E1 16304.303,E2 16304.303} C_VEL
LIN {X 0,Y 389.397,Z 342.882,A -85,B 0,C 180,E1 16300.803,E2 16300.803} C_VEL
LIN {X 0,Y 390.098,Z 343.614,A -85,B 0,C 180,E1 16297.215,E2 16297.215} C_VEL
LIN {X 0,Y 390.513,Z 344.008,A -85,B 0,C 180,E1 16293.523,E2 16293.523} C_VEL
LIN {X 0,Y 390.661,Z 344.116,A -85,B 0,C 180,E1 16289.853,E2 16289.853} C_VEL
LIN {X 0,Y 390.501,Z 344.008,A -85,B 0,C 180,E1 16286.33,E2 16286.33} C_VEL
LIN {X 0,Y 390.086,Z 343.608,A -85,B 0,C 180,E1 16282.637,E2 16282.637} C_VEL
LIN {X 0,Y 389.366,Z 342.851,A -85,B 0,C 180,E1 16279.046,E2 16279.046} C_VEL
LIN {X 0,Y 388.477,Z 341.51,A -85,B 0,C 180,E1 16275.543,E2 16275.543} C_VEL
LIN {X 0,Y 387.392,Z 339.484,A -85,B 0,C 180,E1 16272.114,E2 16272.114} C_VEL
LIN {X 0,Y 386.075,Z 338.516,A -85,B 0,C 180,E1 16268.901,E2 16268.901} C_VEL
LIN {X 0,Y 384.231,Z 337.624,A -85,B 0,C 180,E1 16265.232,E2 16265.232} C_VEL
LIN {X 0,Y 382.375,Z 335.989,A -85,B 0,C 180,E1 16261.753,E2 16261.753} C_VEL
LIN {X 0,Y 380.66,Z 333.363,A -85,B 0,C 180,E1 16258.752,E2 16258.752} C_VEL
LIN {X 0,Y 379.685,Z 331.895,A -85,B 0,C 180,E1 16257.145,E2 16257.145} C_VEL
LIN {X 0,Y 376.985,Z 330.495,A -85,B 0,C 180,E1 16253.363,E2 16253.363} C_VEL
LIN {X 0,Y 374.843,Z 328.447,A -85,B 0,C 180,E1 16250.395,E2 16250.395} C_VEL
LIN {X 0,Y 372.693,Z 324.943,A -85,B 0,C 180,E1 16247.465,E2 16247.465} C_VEL
LIN {X 0,Y 369.511,Z 323.183,A -85,B 0,C 180,E1 16243.743,E2 16243.743} C_VEL
LIN {X 0,Y 367.672,Z 321.278,A -85,B 0,C 180,E1 16241.576,E2 16241.576} C_VEL
LIN {X 0,Y 366.668,Z 320.869,A -85,B 0,C 180,E1 16240.461,E2 16240.461} C_VEL
LIN {X 0,Y 364.558,Z 322.832,A -85,B 0,C 180,E1 16238.577,E2 16238.577} C_VEL
LIN {X 0,Y 362.577,Z 324.514,A -85,B 0,C 180,E1 16236.845,E2 16236.845} C_VEL
LIN {X 0,Y 361.753,Z 324.357,A -85,B 0,C 180,E1 16236.057,E2 16236.057} C_VEL
LIN {X 0,Y 359.316,Z 321.762,A -85,B 0,C 180,E1 16233.433,E2 16233.433} C_VEL
LIN {X 0,Y 357.59,Z 318.827,A -85,B 0,C 180,E1 16231.484,E2 16231.484} C_VEL
LIN {X 0,Y 354.173,Z 316.896,A -85,B 0,C 180,E1 16228.129,E2 16228.129} C_VEL
LIN {X 0,Y 352.037,Z 314.283,A -85,B 0,C 180,E1 16226.119,E2 16226.119} C_VEL
LIN {X 0,Y 350.729,Z 311.993,A -85,B 0,C 180,E1 16224.956,E2 16224.956} C_VEL
LIN {X 0,Y 347.257,Z 309.974,A -85,B 0,C 180,E1 16222.516,E2 16222.516} C_VEL
LIN {X 0,Y 345.143,Z 307.291,A -85,B 0,C 180,E1 16221.052,E2 16221.052} C_VEL
LIN {X 0,Y 343.675,Z 304.936,A -85,B 0,C 180,E1 16220.078,E2 16220.078} C_VEL
LIN {X 0,Y 340.289,Z 302.836,A -85,B 0,C 180,E1 16218.147,E2 16218.147} C_VEL
LIN {X 0,Y 338.332,Z 299.705,A -85,B 0,C 180,E1 16216.835,E2 16216.835} C_VEL
LIN {X 0,Y 337.999,Z 298.368,A -85,B 0,C 180,E1 16216.145,E2 16216.145} C_VEL
LIN {X 0,Y 337.958,Z 298.137,A -85,B 0,C 180,E1 16212.473,E2 16212.473} C_VEL
LIN {X 0,Y 337.955,Z 298.098,A -85,B 0,C 180,E1 16208.164,E2 16208.164} C_VEL
LIN {X 0,Y 337.958,Z 298.084,A -85,B 0,C 180,E1 16203.902,E2 16203.902} C_VEL
LIN {X 0,Y 337.97,Z 298.12,A -85,B 0,C 180,E1 16199.661,E2 16199.661} C_VEL
LIN {X 0,Y 337.974,Z 298.101,A -85,B 0,C 180,E1 16195.419,E2 16195.419} C_VEL
LIN {X 0,Y 337.979,Z 298.082,A -85,B 0,C 180,E1 16191.151,E2 16191.151} C_VEL
LIN {X 0,Y 337.969,Z 298.105,A -85,B 0,C 180,E1 16186.832,E2 16186.832} C_VEL
LIN {X 0,Y 337.978,Z 298.332,A -85,B 0,C 180,E1 16184.383,E2 16184.383} C_VEL
LIN {X 0,Y 338.358,Z 299.799,A -85,B 0,C 180,E1 16183.564,E2 16183.564} C_VEL
LIN {X 0,Y 340.277,Z 302.853,A -85,B 0,C 180,E1 16182.295,E2 16182.295} C_VEL
LIN {X 0,Y 343.953,Z 305.374,A -85,B 0,C 180,E1 16180.337,E2 16180.337} C_VEL
LIN {X 0,Y 345.917,Z 308.758,A -85,B 0,C 180,E1 16179.263,E2 16179.263} C_VEL
LIN {X 0,Y 349.141,Z 311.272,A -85,B 0,C 180,E1 16177.789,E2 16177.789} C_VEL
LIN {X 0,Y 352.173,Z 315.709,A -85,B 0,C 180,E1 16176.402,E2 16176.402} C_VEL
LIN {X 0,Y 354.804,Z 317.984,A -85,B 0,C 180,E1 16175.35,E2 16175.35} C_VEL
LIN {X 0,Y 357.79,Z 322.061,A -85,B 0,C 180,E1 16174.154,E2 16174.154} C_VEL
LIN {X 0,Y 359.896,Z 324.173,A -85,B 0,C 180,E1 16173.386,E2 16173.386} C_VEL
LIN {X 0,Y 363.445,Z 328.627,A -85,B 0,C 180,E1 16172.116,E2 16172.116} C_VEL
LIN {X 0,Y 370.332,Z 338.45,A -85,B 0,C 180,E1 16169.811,E2 16169.811} C_VEL
LIN {X 0,Y 375.475,Z 346.185,A -85,B 0,C 180,E1 16168.225,E2 16168.225} C_VEL
LIN {X 0,Y 383.471,Z 358.76,A -85,B 0,C 180,E1 16165.949,E2 16165.949} C_VEL
LIN {X 0,Y 391.872,Z 373.091,A -85,B 0,C 180,E1 16163.75,E2 16163.75} C_VEL
LIN {X 0,Y 399.842,Z 387.894,A -85,B 0,C 180,E1 16161.811,E2 16161.811} C_VEL
LIN {X 0,Y 389.704,Z 598.266,A -85,B 0,C 180,E1 16157.719,E2 16157.719} C_VEL
LIN {X 0,Y 387.993,Z 617.932,A -85,B 0,C 180,E1 16157.218,E2 16157.218} C_VEL
LIN {X 0,Y 385.009,Z 641.13,A -85,B 0,C 180,E1 16156.384,E2 16156.384} C_VEL
LIN {X 0,Y 382.119,Z 658.832,A -85,B 0,C 180,E1 16155.534,E2 16155.534} C_VEL
LIN {X 0,Y 379.013,Z 675.296,A -85,B 0,C 180,E1 16154.564,E2 16154.564} C_VEL
LIN {X 0,Y 374.841,Z 694.851,A -85,B 0,C 180,E1 16153.171,E2 16153.171} C_VEL
LIN {X 0,Y 370.058,Z 714.266,A -85,B 0,C 180,E1 16151.448,E2 16151.448} C_VEL
LIN {X 0,Y 366.099,Z 729.237,A -85,B 0,C 180,E1 16149.875,E2 16149.875} C_VEL
LIN {X 0,Y 361.383,Z 746.185,A -85,B 0,C 180,E1 16147.794,E2 16147.794} C_VEL
LIN {X 0,Y 356.411,Z 762.996,A -85,B 0,C 180,E1 16145.302,E2 16145.302} C_VEL
LIN {X 0,Y 352.431,Z 776.231,A -85,B 0,C 180,E1 16143.004,E2 16143.004} C_VEL
LIN {X 0,Y 348.288,Z 790.311,A -85,B 0,C 180,E1 16140.157,E2 16140.157} C_VEL
LIN {X 0,Y 344.53,Z 803.185,A -85,B 0,C 180,E1 16137.009,E2 16137.009} C_VEL
LIN {X 0,Y 341.835,Z 813.212,A -85,B 0,C 180,E1 16134.134,E2 16134.134} C_VEL
LIN {X 0,Y 339.316,Z 823.741,A -85,B 0,C 180,E1 16130.527,E2 16130.527} C_VEL
LIN {X 0,Y 337.729,Z 831.546,A -85,B 0,C 180,E1 16127.22,E2 16127.22} C_VEL
LIN {X 0,Y 336.769,Z 837.605,A -85,B 0,C 180,E1 16124.09,E2 16124.09} C_VEL
LIN {X 0,Y 336.164,Z 843.305,A -85,B 0,C 180,E1 16120.28,E2 16120.28} C_VEL
LIN {X 0,Y 335.98,Z 846.683,A -85,B 0,C 180,E1 16117.008,E2 16117.008} C_VEL
LIN {X 0,Y 335.942,Z 848.635,A -85,B 0,C 180,E1 16114.096,E2 16114.096} C_VEL
LIN {X 0,Y 335.946,Z 849.565,A -85,B 0,C 180,E1 16111.194,E2 16111.194} C_VEL
LIN {X 0,Y 335.942,Z 849.482,A -85,B 0,C 180,E1 16108.295,E2 16108.295} C_VEL
LIN {X 0,Y 335.946,Z 848.136,A -85,B 0,C 180,E1 16104.878,E2 16104.878} C_VEL
LIN {X 0,Y 336.044,Z 845.057,A -85,B 0,C 180,E1 16101.272,E2 16101.272} C_VEL
LIN {X 0,Y 336.349,Z 841.157,A -85,B 0,C 180,E1 16098.164,E2 16098.164} C_VEL
LIN {X 0,Y 336.994,Z 836.052,A -85,B 0,C 180,E1 16095.041,E2 16095.041} C_VEL
LIN {X 0,Y 338.323,Z 828.511,A -85,B 0,C 180,E1 16091.387,E2 16091.387} C_VEL
LIN {X 0,Y 340.184,Z 819.901,A -85,B 0,C 180,E1 16088.083,E2 16088.083} C_VEL
LIN {X 0,Y 342.457,Z 810.822,A -85,B 0,C 180,E1 16085.139,E2 16085.139} C_VEL
LIN {X 0,Y 345.768,Z 798.951,A -85,B 0,C 180,E1 16081.879,E2 16081.879} C_VEL
LIN {X 0,Y 349.42,Z 786.305,A -85,B 0,C 180,E1 16078.999,E2 16078.999} C_VEL
LIN {X 0,Y 352.976,Z 774.442,A -85,B 0,C 180,E1 16076.666,E2 16076.666} C_VEL
LIN {X 0,Y 357.644,Z 759.006,A -85,B 0,C 180,E1 16074.05,E2 16074.05} C_VEL
LIN {X 0,Y 362.481,Z 742.224,A -85,B 0,C 180,E1 16071.697,E2 16071.697} C_VEL
LIN {X 0,Y 366.759,Z 726.833,A -85,B 0,C 180,E1 16069.855,E2 16069.855} C_VEL
LIN {X 0,Y 371.758,Z 707.723,A -85,B 0,C 180,E1 16067.929,E2 16067.929} C_VEL
LIN {X 0,Y 375.894,Z 689.913,A -85,B 0,C 180,E1 16066.456,E2 16066.456} C_VEL
LIN {X 0,Y 379.461,Z 673.029,A -85,B 0,C 180,E1 16065.291,E2 16065.291} C_VEL
LIN {X 0,Y 383.305,Z 652.189,A -85,B 0,C 180,E1 16064.113,E2 16064.113} C_VEL
LIN {X 0,Y 386.407,Z 630.896,A -85,B 0,C 180,E1 16063.212,E2 16063.212} C_VEL
LIN {X 0,Y 388.598,Z 611.999,A -85,B 0,C 180,E1 16062.614,E2 16062.614} C_VEL
LIN {X 0,Y 390.381,Z 585.984,A -85,B 0,C 180,E1 16062.025,E2 16062.025} C_VEL
LIN {X 0,Y 399.824,Z 387.859,A -85,B 0,C 180,E1 16058.185,E2 16058.185} C_VEL
LIN {X 0,Y 391.056,Z 371.606,A -85,B 0,C 180,E1 16056.042,E2 16056.042} C_VEL
LIN {X 0,Y 380.968,Z 354.578,A -85,B 0,C 180,E1 16053.356,E2 16053.356} C_VEL
LIN {X 0,Y 372.214,Z 341.171,A -85,B 0,C 180,E1 16050.779,E2 16050.779} C_VEL
LIN {X 0,Y 363.867,Z 329.089,A -85,B 0,C 180,E1 16048.027,E2 16048.027} C_VEL
LIN {X 0,Y 359.896,Z 324.173,A -85,B 0,C 180,E1 16046.614,E2 16046.614} C_VEL
LIN {X 0,Y 355.513,Z 319.207,A -85,B 0,C 180,E1 16044.952,E2 16044.952} C_VEL
LIN {X 0,Y 354.246,Z 317.354,A -85,B 0,C 180,E1 16044.425,E2 16044.425} C_VEL
LIN {X 0,Y 351.026,Z 314.361,A -85,B 0,C 180,E1 16043.102,E2 16043.102} C_VEL
LIN {X 0,Y 349.14,Z 311.281,A -85,B 0,C 180,E1 16042.211,E2 16042.211} C_VEL
LIN {X 0,Y 345.917,Z 308.757,A -85,B 0,C 180,E1 16040.737,E2 16040.737} C_VEL
LIN {X 0,Y 343.43,Z 304.781,A -85,B 0,C 180,E1 16039.384,E2 16039.384} C_VEL
LIN {X 0,Y 340.006,Z 302.558,A -85,B 0,C 180,E1 16037.543,E2 16037.543} C_VEL
LIN {X 0,Y 338.068,Z 298.83,A -85,B 0,C 180,E1 16036.017,E2 16036.017} C_VEL
LIN {X 0,Y 337.991,Z 298.114,A -85,B 0,C 180,E1 16034.914,E2 16034.914} C_VEL
LIN {X 0,Y 337.966,Z 298.098,A -85,B 0,C 180,E1 16030.569,E2 16030.569} C_VEL
LIN {X 0,Y 337.961,Z 298.131,A -85,B 0,C 180,E1 16026.265,E2 16026.265} C_VEL
LIN {X 0,Y 337.951,Z 298.088,A -85,B 0,C 180,E1 16022.035,E2 16022.035} C_VEL
LIN {X 0,Y 337.949,Z 298.094,A -85,B 0,C 180,E1 16017.796,E2 16017.796} C_VEL
LIN {X 0,Y 337.96,Z 298.139,A -85,B 0,C 180,E1 16013.374,E2 16013.374} C_VEL
LIN {X 0,Y 337.965,Z 298.095,A -85,B 0,C 180,E1 16009.086,E2 16009.086} C_VEL
LIN {X 0,Y 337.971,Z 298.094,A -85,B 0,C 180,E1 16004.91,E2 16004.91} C_VEL
LIN {X 0,Y 338.032,Z 298.571,A -85,B 0,C 180,E1 16003.68,E2 16003.68} C_VEL
LIN {X 0,Y 338.628,Z 300.424,A -85,B 0,C 180,E1 16002.915,E2 16002.915} C_VEL
LIN {X 0,Y 340.85,Z 303.352,A -85,B 0,C 180,E1 16001.53,E2 16001.53} C_VEL
LIN {X 0,Y 344.184,Z 305.48,A -85,B 0,C 180,E1 15999.598,E2 15999.598} C_VEL
LIN {X 0,Y 346.414,Z 309.178,A -85,B 0,C 180,E1 15998.051,E2 15998.051} C_VEL
LIN {X 0,Y 349.36,Z 311.32,A -85,B 0,C 180,E1 15996.021,E2 15996.021} C_VEL
LIN {X 0,Y 351.111,Z 312.496,A -85,B 0,C 180,E1 15994.713,E2 15994.713} C_VEL
LIN {X 0,Y 352.931,Z 315.585,A -85,B 0,C 180,E1 15993.046,E2 15993.046} C_VEL
LIN {X 0,Y 355.201,Z 317.628,A -85,B 0,C 180,E1 15990.858,E2 15990.858} C_VEL
LIN {X 0,Y 357.981,Z 319.247,A -85,B 0,C 180,E1 15988.11,E2 15988.11} C_VEL
LIN {X 0,Y 360.132,Z 322.846,A -85,B 0,C 180,E1 15985.695,E2 15985.695} C_VEL
LIN {X 0,Y 362.859,Z 325.01,A -85,B 0,C 180,E1 15982.78,E2 15982.78} C_VEL
LIN {X 0,Y 364.922,Z 326.211,A -85,B 0,C 180,E1 15980.591,E2 15980.591} C_VEL
LIN {X 0,Y 367.1,Z 329.843,A -85,B 0,C 180,E1 15977.931,E2 15977.931} C_VEL
LIN {X 0,Y 369.714,Z 331.907,A -85,B 0,C 180,E1 15974.883,E2 15974.883} C_VEL
LIN {X 0,Y 371.951,Z 333.21,A -85,B 0,C 180,E1 15972.223,E2 15972.223} C_VEL
LIN {X 0,Y 373.836,Z 336.43,A -85,B 0,C 180,E1 15969.621,E2 15969.621} C_VEL
LIN {X 0,Y 376.067,Z 338.496,A -85,B 0,C 180,E1 15966.551,E2 15966.551} C_VEL
LIN {X 0,Y 378.764,Z 339.911,A -85,B 0,C 180,E1 15962.761,E2 15962.761} C_VEL
LIN {X 0,Y 380.799,Z 343.293,A -85,B 0,C 180,E1 15959.233,E2 15959.233} C_VEL
LIN {X 0,Y 382.677,Z 345.139,A -85,B 0,C 180,E1 15955.87,E2 15955.87} C_VEL
LIN {X 0,Y 384.443,Z 346.179,A -85,B 0,C 180,E1 15952.477,E2 15952.477} C_VEL
LIN {X 0,Y 386.076,Z 347.053,A -85,B 0,C 180,E1 15948.888,E2 15948.888} C_VEL
LIN {X 0,Y 387.05,Z 348.726,A -85,B 0,C 180,E1 15945.892,E2 15945.892} C_VEL
LIN {X 0,Y 388.052,Z 350.348,A -85,B 0,C 180,E1 15942.348,E2 15942.348} C_VEL
LIN {X 0,Y 388.824,Z 351.288,A -85,B 0,C 180,E1 15938.726,E2 15938.726} C_VEL
LIN {X 0,Y 389.384,Z 351.796,A -85,B 0,C 180,E1 15935.304,E2 15935.304} C_VEL
LIN {X 0,Y 389.635,Z 352.029,A -85,B 0,C 180,E1 15931.617,E2 15931.617} C_VEL
LIN {X 0,Y 389.646,Z 352.038,A -85,B 0,C 180,E1 15928.088,E2 15928.088} C_VEL
LIN {X 0,Y 389.33,Z 351.785,A -85,B 0,C 180,E1 15924.4,E2 15924.4} C_VEL
LIN {X 0,Y 388.773,Z 351.22,A -85,B 0,C 180,E1 15920.825,E2 15920.825} C_VEL
LIN {X 0,Y 387.949,Z 350.199,A -85,B 0,C 180,E1 15917.195,E2 15917.195} C_VEL
LIN {X 0,Y 386.97,Z 348.485,A -85,B 0,C 180,E1 15913.797,E2 15913.797} C_VEL
LIN {X 0,Y 385.922,Z 346.947,A -85,B 0,C 180,E1 15910.79,E2 15910.79} C_VEL
LIN {X 0,Y 384.357,Z 346.148,A -85,B 0,C 180,E1 15907.357,E2 15907.357} C_VEL
LIN {X 0,Y 382.486,Z 344.985,A -85,B 0,C 180,E1 15903.719,E2 15903.719} C_VEL
LIN {X 0,Y 380.614,Z 342.997,A -85,B 0,C 180,E1 15900.403,E2 15900.403} C_VEL
LIN {X 0,Y 378.764,Z 339.911,A -85,B 0,C 180,E1 15897.239,E2 15897.239} C_VEL
LIN {X 0,Y 376.066,Z 338.495,A -85,B 0,C 180,E1 15893.449,E2 15893.449} C_VEL
LIN {X 0,Y 373.836,Z 336.43,A -85,B 0,C 180,E1 15890.379,E2 15890.379} C_VEL
LIN {X 0,Y 372.192,Z 333.594,A -85,B 0,C 180,E1 15888.085,E2 15888.085} C_VEL
LIN {X 0,Y 371.027,Z 332.515,A -85,B 0,C 180,E1 15886.594,E2 15886.594} C_VEL
LIN {X 0,Y 368.142,Z 330.828,A -85,B 0,C 180,E1 15883.293,E2 15883.293} C_VEL
LIN {X 0,Y 366.115,Z 328.394,A -85,B 0,C 180,E1 15880.846,E2 15880.846} C_VEL
LIN {X 0,Y 364.513,Z 325.755,A -85,B 0,C 180,E1 15878.913,E2 15878.913} C_VEL
LIN {X 0,Y 361.753,Z 324.357,A -85,B 0,C 180,E1 15876.057,E2 15876.057} C_VEL
LIN {X 0,Y 360.259,Z 324.227,A -85,B 0,C 180,E1 15874.579,E2 15874.579} C_VEL
LIN {X 0,Y 356.366,Z 326.437,A -85,B 0,C 180,E1 15871.174,E2 15871.174} C_VEL
LIN {X 0,Y 355.6,Z 326.344,A -85,B 0,C 180,E1 15870.467,E2 15870.467} C_VEL
LIN {X 0,Y 352.559,Z 324.302,A -85,B 0,C 180,E1 15867.533,E2 15867.533} C_VEL
LIN {X 0,Y 350.432,Z 321.589,A -85,B 0,C 180,E1 15865.632,E2 15865.632} C_VEL
LIN {X 0,Y 349.363,Z 319.738,A -85,B 0,C 180,E1 15864.698,E2 15864.698} C_VEL
LIN {X 0,Y 345.843,Z 317.693,A -85,B 0,C 180,E1 15862.255,E2 15862.255} C_VEL
LIN {X 0,Y 343.53,Z 314.873,A -85,B 0,C 180,E1 15860.709,E2 15860.709} C_VEL
LIN {X 0,Y 342.208,Z 312.673,A -85,B 0,C 180,E1 15859.811,E2 15859.811} C_VEL
LIN {X 0,Y 338.78,Z 310.526,A -85,B 0,C 180,E1 15857.875,E2 15857.875} C_VEL
LIN {X 0,Y 336.509,Z 306.968,A -85,B 0,C 180,E1 15856.351,E2 15856.351} C_VEL
LIN {X 0,Y 335.625,Z 305.798,A -85,B 0,C 180,E1 15855.73,E2 15855.73} C_VEL
LIN {X 0,Y 331.988,Z 303.431,A -85,B 0,C 180,E1 15853.055,E2 15853.055} C_VEL
LIN {X 0,Y 330.337,Z 300.464,A -85,B 0,C 180,E1 15851.368,E2 15851.368} C_VEL
LIN {X 0,Y 330.037,Z 299.173,A -85,B 0,C 180,E1 15849.944,E2 15849.944} C_VEL
LIN {X 0,Y 330.034,Z 299.102,A -85,B 0,C 180,E1 15845.738,E2 15845.738} C_VEL
LIN {X 0,Y 330.045,Z 299.093,A -85,B 0,C 180,E1 15841.389,E2 15841.389} C_VEL
LIN {X 0,Y 330.031,Z 299.069,A -85,B 0,C 180,E1 15837.048,E2 15837.048} C_VEL
LIN {X 0,Y 330.02,Z 299.089,A -85,B 0,C 180,E1 15832.689,E2 15832.689} C_VEL
LIN {X 0,Y 330.054,Z 299.415,A -85,B 0,C 180,E1 15830.057,E2 15830.057} C_VEL
LIN {X 0,Y 330.44,Z 300.81,A -85,B 0,C 180,E1 15828.922,E2 15828.922} C_VEL
LIN {X 0,Y 332.081,Z 303.528,A -85,B 0,C 180,E1 15827.303,E2 15827.303} C_VEL
LIN {X 0,Y 336.224,Z 306.379,A -85,B 0,C 180,E1 15824.299,E2 15824.299} C_VEL
LIN {X 0,Y 338.498,Z 310.255,A -85,B 0,C 180,E1 15822.731,E2 15822.731} C_VEL
LIN {X 0,Y 342.074,Z 312.878,A -85,B 0,C 180,E1 15820.758,E2 15820.758} C_VEL
LIN {X 0,Y 344.474,Z 316.668,A -85,B 0,C 180,E1 15819.439,E2 15819.439} C_VEL
LIN {X 0,Y 347.557,Z 319.354,A -85,B 0,C 180,E1 15817.994,E2 15817.994} C_VEL
LIN {X 0,Y 350.32,Z 323.254,A -85,B 0,C 180,E1 15816.716,E2 15816.716} C_VEL
LIN {X 0,Y 352.712,Z 325.493,A -85,B 0,C 180,E1 15815.73,E2 15815.73} C_VEL
LIN {X 0,Y 356.059,Z 329.802,A -85,B 0,C 180,E1 15814.377,E2 15814.377} C_VEL
LIN {X 0,Y 357.726,Z 331.67,A -85,B 0,C 180,E1 15813.748,E2 15813.748} C_VEL
LIN {X 0,Y 363.076,Z 338.579,A -85,B 0,C 180,E1 15811.817,E2 15811.817} C_VEL
LIN {X 0,Y 371.647,Z 351.458,A -85,B 0,C 180,E1 15808.989,E2 15808.989} C_VEL
LIN {X 0,Y 380.281,Z 365.345,A -85,B 0,C 180,E1 15806.441,E2 15806.441} C_VEL
LIN {X 0,Y 389.052,Z 380.635,A -85,B 0,C 180,E1 15804.084,E2 15804.084} C_VEL
LIN {X 0,Y 394.728,Z 391.641,A -85,B 0,C 180,E1 15802.647,E2 15802.647} C_VEL
LIN {X 0,Y 384.216,Z 599.847,A -85,B 0,C 180,E1 15798.564,E2 15798.564} C_VEL
LIN {X 0,Y 382.15,Z 621.931,A -85,B 0,C 180,E1 15797.976,E2 15797.976} C_VEL
LIN {X 0,Y 379.304,Z 642.035,A -85,B 0,C 180,E1 15797.214,E2 15797.214} C_VEL
LIN {X 0,Y 376.298,Z 659.666,A -85,B 0,C 180,E1 15796.353,E2 15796.353} C_VEL
LIN {X 0,Y 372.815,Z 677.31,A -85,B 0,C 180,E1 15795.291,E2 15795.291} C_VEL
LIN {X 0,Y 367.82,Z 699.019,A -85,B 0,C 180,E1 15793.665,E2 15793.665} C_VEL
LIN {X 0,Y 363.552,Z 715.555,A -85,B 0,C 180,E1 15792.148,E2 15792.148} C_VEL
LIN {X 0,Y 359.026,Z 731.894,A -85,B 0,C 180,E1 15790.381,E2 15790.381} C_VEL
LIN {X 0,Y 353.507,Z 750.465,A -85,B 0,C 180,E1 15787.963,E2 15787.963} C_VEL
LIN {X 0,Y 349.37,Z 763.776,A -85,B 0,C 180,E1 15785.913,E2 15785.913} C_VEL
LIN {X 0,Y 345.239,Z 776.869,A -85,B 0,C 180,E1 15783.583,E2 15783.583} C_VEL
LIN {X 0,Y 340.666,Z 791.502,A -85,B 0,C 180,E1 15780.514,E2 15780.514} C_VEL
LIN {X 0,Y 337.068,Z 803.239,A -85,B 0,C 180,E1 15777.564,E2 15777.564} C_VEL
LIN {X 0,Y 334.172,Z 813.405,A -85,B 0,C 180,E1 15774.575,E2 15774.575} C_VEL
LIN {X 0,Y 331.382,Z 824.352,A -85,B 0,C 180,E1 15770.671,E2 15770.671} C_VEL
LIN {X 0,Y 329.892,Z 831.291,A -85,B 0,C 180,E1 15767.643,E2 15767.643} C_VEL
LIN {X 0,Y 328.851,Z 837.351,A -85,B 0,C 180,E1 15764.437,E2 15764.437} C_VEL
LIN {X 0,Y 328.19,Z 843.053,A -85,B 0,C 180,E1 15760.532,E2 15760.532} C_VEL
LIN {X 0,Y 327.989,Z 846.433,A -85,B 0,C 180,E1 15757.18,E2 15757.18} C_VEL
LIN {X 0,Y 327.945,Z 848.386,A -85,B 0,C 180,E1 15754.196,E2 15754.196} C_VEL
LIN {X 0,Y 327.95,Z 849.317,A -85,B 0,C 180,E1 15751.223,E2 15751.223} C_VEL
LIN {X 0,Y 327.945,Z 849.234,A -85,B 0,C 180,E1 15748.253,E2 15748.253} C_VEL
LIN {X 0,Y 327.948,Z 847.886,A -85,B 0,C 180,E1 15744.752,E2 15744.752} C_VEL
LIN {X 0,Y 328.052,Z 844.806,A -85,B 0,C 180,E1 15741.058,E2 15741.058} C_VEL
LIN {X 0,Y 328.392,Z 840.905,A -85,B 0,C 180,E1 15737.873,E2 15737.873} C_VEL
LIN {X 0,Y 329.091,Z 835.798,A -85,B 0,C 180,E1 15734.673,E2 15734.673} C_VEL
LIN {X 0,Y 330.53,Z 828.255,A -85,B 0,C 180,E1 15730.932,E2 15730.932} C_VEL
LIN {X 0,Y 332.522,Z 819.645,A -85,B 0,C 180,E1 15727.551,E2 15727.551} C_VEL
LIN {X 0,Y 334.953,Z 810.565,A -85,B 0,C 180,E1 15724.543,E2 15724.543} C_VEL
LIN {X 0,Y 338.472,Z 798.693,A -85,B 0,C 180,E1 15721.217,E2 15721.217} C_VEL
LIN {X 0,Y 342.341,Z 786.048,A -85,B 0,C 180,E1 15718.284,E2 15718.284} C_VEL
LIN {X 0,Y 346.092,Z 774.185,A -85,B 0,C 180,E1 15715.913,E2 15715.913} C_VEL
LIN {X 0,Y 350.989,Z 758.75,A -85,B 0,C 180,E1 15713.258,E2 15713.258} C_VEL
LIN {X 0,Y 355.985,Z 742.229,A -85,B 0,C 180,E1 15710.91,E2 15710.91} C_VEL
LIN {X 0,Y 360.331,Z 727.266,A -85,B 0,C 180,E1 15709.092,E2 15709.092} C_VEL
LIN {X 0,Y 365.257,Z 709.385,A -85,B 0,C 180,E1 15707.245,E2 15707.245} C_VEL
LIN {X 0,Y 370.036,Z 689.66,A -85,B 0,C 180,E1 15705.588,E2 15705.588} C_VEL
LIN {X 0,Y 373.739,Z 672.777,A -85,B 0,C 180,E1 15704.416,E2 15704.416} C_VEL
LIN {X 0,Y 377.748,Z 651.813,A -85,B 0,C 180,E1 15703.227,E2 15703.227} C_VEL
LIN {X 0,Y 380.939,Z 630.674,A -85,B 0,C 180,E1 15702.331,E2 15702.331} C_VEL
LIN {X 0,Y 383.189,Z 611.891,A -85,B 0,C 180,E1 15701.734,E2 15701.734} C_VEL
LIN {X 0,Y 385.012,Z 586.5,A -85,B 0,C 180,E1 15701.151,E2 15701.151} C_VEL
LIN {X 0,Y 394.741,Z 391.367,A -85,B 0,C 180,E1 15697.347,E2 15697.347} C_VEL
LIN {X 0,Y 386.565,Z 376.248,A -85,B 0,C 180,E1 15695.271,E2 15695.271} C_VEL
LIN {X 0,Y 377.352,Z 360.415,A -85,B 0,C 180,E1 15692.72,E2 15692.72} C_VEL
LIN {X 0,Y 369.219,Z 347.748,A -85,B 0,C 180,E1 15690.245,E2 15690.245} C_VEL
LIN {X 0,Y 361.24,Z 335.987,A -85,B 0,C 180,E1 15687.531,E2 15687.531} C_VEL
LIN {X 0,Y 357.349,Z 331.057,A -85,B 0,C 180,E1 15686.103,E2 15686.103} C_VEL
LIN {X 0,Y 353.239,Z 326.362,A -85,B 0,C 180,E1 15684.499,E2 15684.499} C_VEL
LIN {X 0,Y 351.981,Z 324.661,A -85,B 0,C 180,E1 15683.967,E2 15683.967} C_VEL
LIN {X 0,Y 348.597,Z 321.138,A -85,B 0,C 180,E1 15682.514,E2 15682.514} C_VEL
LIN {X 0,Y 347.15,Z 318.792,A -85,B 0,C 180,E1 15681.811,E2 15681.811} C_VEL
LIN {X 0,Y 343.856,Z 315.923,A -85,B 0,C 180,E1 15680.244,E2 15680.244} C_VEL
LIN {X 0,Y 341.866,Z 312.527,A -85,B 0,C 180,E1 15679.121,E2 15679.121} C_VEL
LIN {X 0,Y 338.499,Z 310.252,A -85,B 0,C 180,E1 15677.269,E2 15677.269} C_VEL
LIN {X 0,Y 335.858,Z 306.023,A -85,B 0,C 180,E1 15675.453,E2 15675.453} C_VEL
LIN {X 0,Y 331.884,Z 303.317,A -85,B 0,C 180,E1 15672.528,E2 15672.528} C_VEL
LIN {X 0,Y 330.156,Z 299.855,A -85,B 0,C 180,E1 15670.469,E2 15670.469} C_VEL
LIN {X 0,Y 330.043,Z 299.113,A -85,B 0,C 180,E1 15668.712,E2 15668.712} C_VEL
LIN {X 0,Y 330.032,Z 299.087,A -85,B 0,C 180,E1 15664.518,E2 15664.518} C_VEL
LIN {X 0,Y 330.022,Z 299.113,A -85,B 0,C 180,E1 15660.174,E2 15660.174} C_VEL
LIN {X 0,Y 330.013,Z 299.075,A -85,B 0,C 180,E1 15655.83,E2 15655.83} C_VEL
LIN {X 0,Y 330.014,Z 299.079,A -85,B 0,C 180,E1 15651.462,E2 15651.462} C_VEL
LIN {X 0,Y 330.104,Z 299.628,A -85,B 0,C 180,E1 15649.353,E2 15649.353} C_VEL
LIN {X 0,Y 330.581,Z 301.16,A -85,B 0,C 180,E1 15648.308,E2 15648.308} C_VEL
LIN {X 0,Y 332.391,Z 303.828,A -85,B 0,C 180,E1 15646.607,E2 15646.607} C_VEL
LIN {X 0,Y 336.296,Z 306.433,A -85,B 0,C 180,E1 15643.815,E2 15643.815} C_VEL
LIN {X 0,Y 338.379,Z 310.086,A -85,B 0,C 180,E1 15642.37,E2 15642.37} C_VEL
LIN {X 0,Y 341.325,Z 312.28,A -85,B 0,C 180,E1 15640.67,E2 15640.67} C_VEL
LIN {X 0,Y 342.637,Z 313.236,A -85,B 0,C 180,E1 15639.903,E2 15639.903} C_VEL
LIN {X 0,Y 344.971,Z 316.888,A -85,B 0,C 180,E1 15638.313,E2 15638.313} C_VEL
LIN {X 0,Y 347.987,Z 319.104,A -85,B 0,C 180,E1 15636.281,E2 15636.281} C_VEL
LIN {X 0,Y 349.76,Z 320.269,A -85,B 0,C 180,E1 15634.983,E2 15634.983} C_VEL
LIN {X 0,Y 351.623,Z 323.321,A -85,B 0,C 180,E1 15633.302,E2 15633.302} C_VEL
LIN {X 0,Y 353.966,Z 325.43,A -85,B 0,C 180,E1 15631.117,E2 15631.117} C_VEL
LIN {X 0,Y 356.876,Z 327.185,A -85,B 0,C 180,E1 15628.216,E2 15628.216} C_VEL
LIN {X 0,Y 358.885,Z 330.605,A -85,B 0,C 180,E1 15625.945,E2 15625.945} C_VEL
LIN {X 0,Y 361.722,Z 332.883,A -85,B 0,C 180,E1 15622.945,E2 15622.945} C_VEL
LIN {X 0,Y 363.762,Z 334.04,A -85,B 0,C 180,E1 15620.788,E2 15620.788} C_VEL
LIN {X 0,Y 365.885,Z 337.611,A -85,B 0,C 180,E1 15618.181,E2 15618.181} C_VEL
LIN {X 0,Y 368.682,Z 339.831,A -85,B 0,C 180,E1 15614.942,E2 15614.942} C_VEL
LIN {X 0,Y 370.837,Z 341.074,A -85,B 0,C 180,E1 15612.374,E2 15612.374} C_VEL
LIN {X 0,Y 372.648,Z 344.194,A -85,B 0,C 180,E1 15609.882,E2 15609.882} C_VEL
LIN {X 0,Y 374.864,Z 346.296,A -85,B 0,C 180,E1 15606.853,E2 15606.853} C_VEL
LIN {X 0,Y 377.59,Z 347.701,A -85,B 0,C 180,E1 15603.057,E2 15603.057} C_VEL
LIN {X 0,Y 378.628,Z 349.355,A -85,B 0,C 180,E1 15601.346,E2 15601.346} C_VEL
LIN {X 0,Y 380.414,Z 351.919,A -85,B 0,C 180,E1 15598.235,E2 15598.235} C_VEL
LIN {X 0,Y 382.241,Z 353.502,A -85,B 0,C 180,E1 15594.814,E2 15594.814} C_VEL
LIN {X 0,Y 384.064,Z 354.374,A -85,B 0,C 180,E1 15591.214,E2 15591.214} C_VEL
LIN {X 0,Y 385.349,Z 355.271,A -85,B 0,C 180,E1 15588.141,E2 15588.141} C_VEL
LIN {X 0,Y 386.489,Z 357.341,A -85,B 0,C 180,E1 15584.637,E2 15584.637} C_VEL
LIN {X 0,Y 387.396,Z 358.723,A -85,B 0,C 180,E1 15581.01,E2 15581.01} C_VEL
LIN {X 0,Y 388.125,Z 359.487,A -85,B 0,C 180,E1 15577.4,E2 15577.4} C_VEL
LIN {X 0,Y 388.542,Z 359.887,A -85,B 0,C 180,E1 15573.689,E2 15573.689} C_VEL
LIN {X 0,Y 388.711,Z 359.997,A -85,B 0,C 180,E1 15570.147,E2 15570.147} C_VEL
LIN {X 0,Y 388.569,Z 359.888,A -85,B 0,C 180,E1 15566.607,E2 15566.607} C_VEL
LIN {X 0,Y 388.17,Z 359.523,A -85,B 0,C 180,E1 15563.047,E2 15563.047} C_VEL
LIN {X 0,Y 387.494,Z 358.824,A -85,B 0,C 180,E1 15559.444,E2 15559.444} C_VEL
LIN {X 0,Y 386.604,Z 357.624,A -85,B 0,C 180,E1 15555.893,E2 15555.893} C_VEL
LIN {X 0,Y 385.503,Z 355.576,A -85,B 0,C 180,E1 15552.335,E2 15552.335} C_VEL
LIN {X 0,Y 384.375,Z 354.498,A -85,B 0,C 180,E1 15549.442,E2 15549.442} C_VEL
LIN {X 0,Y 382.603,Z 353.672,A -85,B 0,C 180,E1 15545.778,E2 15545.778} C_VEL
LIN {X 0,Y 380.669,Z 352.212,A -85,B 0,C 180,E1 15542.271,E2 15542.271} C_VEL
LIN {X 0,Y 378.936,Z 349.911,A -85,B 0,C 180,E1 15539.211,E2 15539.211} C_VEL
LIN {X 0,Y 377.665,Z 347.77,A -85,B 0,C 180,E1 15537.061,E2 15537.061} C_VEL
LIN {X 0,Y 374.994,Z 346.388,A -85,B 0,C 180,E1 15533.327,E2 15533.327} C_VEL
LIN {X 0,Y 372.804,Z 344.382,A -85,B 0,C 180,E1 15530.33,E2 15530.33} C_VEL
LIN {X 0,Y 371.145,Z 341.631,A -85,B 0,C 180,E1 15528.034,E2 15528.034} C_VEL
LIN {X 0,Y 370.102,Z 340.482,A -85,B 0,C 180,E1 15526.672,E2 15526.672} C_VEL
LIN {X 0,Y 367.186,Z 338.832,A -85,B 0,C 180,E1 15523.33,E2 15523.33} C_VEL
LIN {X 0,Y 365.066,Z 336.396,A -85,B 0,C 180,E1 15520.784,E2 15520.784} C_VEL
LIN {X 0,Y 363.468,Z 333.678,A -85,B 0,C 180,E1 15518.844,E2 15518.844} C_VEL
LIN {X 0,Y 360.328,Z 331.986,A -85,B 0,C 180,E1 15515.609,E2 15515.609} C_VEL
LIN {X 0,Y 358.023,Z 329.376,A -85,B 0,C 180,E1 15513.092,E2 15513.092} C_VEL
LIN {X 0,Y 356.552,Z 326.788,A -85,B 0,C 180,E1 15511.439,E2 15511.439} C_VEL
LIN {X 0,Y 355.6,Z 326.344,A -85,B 0,C 180,E1 15510.467,E2 15510.467} C_VEL
LIN {X 0,Y 354.613,Z 326.929,A -85,B 0,C 180,E1 15509.635,E2 15509.635} C_VEL
LIN {X 0,Y 351.726,Z 331.312,A -85,B 0,C 180,E1 15507.575,E2 15507.575} C_VEL
LIN {X 0,Y 350.661,Z 331.428,A -85,B 0,C 180,E1 15506.747,E2 15506.747} C_VEL
LIN {X 0,Y 348.609,Z 328.447,A -85,B 0,C 180,E1 15504.937,E2 15504.937} C_VEL
LIN {X 0,Y 347.775,Z 327.449,A -85,B 0,C 180,E1 15504.307,E2 15504.307} C_VEL
LIN {X 0,Y 344.273,Z 325.303,A -85,B 0,C 180,E1 15501.913,E2 15501.913} C_VEL
LIN {X 0,Y 341.801,Z 322.254,A -85,B 0,C 180,E1 15500.282,E2 15500.282} C_VEL
LIN {X 0,Y 340.688,Z 320.432,A -85,B 0,C 180,E1 15499.546,E2 15499.546} C_VEL
LIN {X 0,Y 337.146,Z 318.077,A -85,B 0,C 180,E1 15497.518,E2 15497.518} C_VEL
LIN {X 0,Y 334.816,Z 314.353,A -85,B 0,C 180,E1 15495.902,E2 15495.902} C_VEL
LIN {X 0,Y 334.176,Z 313.566,A -85,B 0,C 180,E1 15495.443,E2 15495.443} C_VEL
LIN {X 0,Y 330.628,Z 311.128,A -85,B 0,C 180,E1 15492.754,E2 15492.754} C_VEL
LIN {X 0,Y 328.343,Z 307.247,A -85,B 0,C 180,E1 15490.35,E2 15490.35} C_VEL
LIN {X 0,Y 323.737,Z 304.032,A -85,B 0,C 180,E1 15481.77,E2 15481.77} C_VEL
LIN {X 0,Y 323.948,Z 304.266,A -85,B 0,C 180,E1 15477.523,E2 15477.523} C_VEL
LIN {X 0,Y 328.417,Z 307.322,A -85,B 0,C 180,E1 15470.007,E2 15470.007} C_VEL
LIN {X 0,Y 330.912,Z 311.427,A -85,B 0,C 180,E1 15467.435,E2 15467.435} C_VEL
LIN {X 0,Y 334.703,Z 314.079,A -85,B 0,C 180,E1 15464.626,E2 15464.626} C_VEL
LIN {X 0,Y 336.869,Z 317.798,A -85,B 0,C 180,E1 15463.09,E2 15463.09} C_VEL
LIN {X 0,Y 340.35,Z 320.621,A -85,B 0,C 180,E1 15461.102,E2 15461.102} C_VEL
LIN {X 0,Y 343.196,Z 324.709,A -85,B 0,C 180,E1 15459.537,E2 15459.537} C_VEL
LIN {X 0,Y 345.581,Z 326.819,A -85,B 0,C 180,E1 15458.397,E2 15458.397} C_VEL
LIN {X 0,Y 348.655,Z 330.975,A -85,B 0,C 180,E1 15456.955,E2 15456.955} C_VEL
LIN {X 0,Y 350.641,Z 332.959,A -85,B 0,C 180,E1 15456.114,E2 15456.114} C_VEL
LIN {X 0,Y 354.334,Z 337.532,A -85,B 0,C 180,E1 15454.602,E2 15454.602} C_VEL
LIN {X 0,Y 360.342,Z 345.315,A -85,B 0,C 180,E1 15452.35,E2 15452.35} C_VEL
LIN {X 0,Y 368.746,Z 358.222,A -85,B 0,C 180,E1 15449.487,E2 15449.487} C_VEL
LIN {X 0,Y 376.886,Z 371.543,A -85,B 0,C 180,E1 15447.008,E2 15447.008} C_VEL
LIN {X 0,Y 385.813,Z 387.388,A -85,B 0,C 180,E1 15444.537,E2 15444.537} C_VEL
LIN {X 0,Y 389.703,Z 395.106,A -85,B 0,C 180,E1 15443.514,E2 15443.514} C_VEL
LIN {X 0,Y 378.903,Z 600.216,A -85,B 0,C 180,E1 15439.461,E2 15439.461} C_VEL
LIN {X 0,Y 376.696,Z 622.56,A -85,B 0,C 180,E1 15438.855,E2 15438.855} C_VEL
LIN {X 0,Y 373.656,Z 643.086,A -85,B 0,C 180,E1 15438.062,E2 15438.062} C_VEL
LIN {X 0,Y 370.592,Z 660.308,A -85,B 0,C 180,E1 15437.209,E2 15437.209} C_VEL
LIN {X 0,Y 366.558,Z 679.902,A -85,B 0,C 180,E1 15436.005,E2 15436.005} C_VEL
LIN {X 0,Y 361.74,Z 699.634,A -85,B 0,C 180,E1 15434.48,E2 15434.48} C_VEL
LIN {X 0,Y 357.378,Z 715.858,A -85,B 0,C 180,E1 15432.971,E2 15432.971} C_VEL
LIN {X 0,Y 352.364,Z 733.207,A -85,B 0,C 180,E1 15431.062,E2 15431.062} C_VEL
LIN {X 0,Y 346.86,Z 750.762,A -85,B 0,C 180,E1 15428.719,E2 15428.719} C_VEL
LIN {X 0,Y 342.397,Z 764.474,A -85,B 0,C 180,E1 15426.562,E2 15426.562} C_VEL
LIN {X 0,Y 337.514,Z 779.297,A -85,B 0,C 180,E1 15423.843,E2 15423.843} C_VEL
LIN {X 0,Y 332.817,Z 793.402,A -85,B 0,C 180,E1 15420.711,E2 15420.711} C_VEL
LIN {X 0,Y 329.337,Z 804.264,A -85,B 0,C 180,E1 15417.874,E2 15417.874} C_VEL
LIN {X 0,Y 325.887,Z 815.893,A -85,B 0,C 180,E1 15414.275,E2 15414.275} C_VEL
LIN {X 0,Y 323.45,Z 824.964,A -85,B 0,C 180,E1 15410.823,E2 15410.823} C_VEL
LIN {X 0,Y 321.914,Z 831.778,A -85,B 0,C 180,E1 15407.721,E2 15407.721} C_VEL
LIN {X 0,Y 320.719,Z 838.63,A -85,B 0,C 180,E1 15403.889,E2 15403.889} C_VEL
LIN {X 0,Y 320.144,Z 843.581,A -85,B 0,C 180,E1 15400.072,E2 15400.072} C_VEL
LIN {X 0,Y 319.98,Z 846.46,A -85,B 0,C 180,E1 15397,E2 15397} C_VEL
LIN {X 0,Y 319.944,Z 848.302,A -85,B 0,C 180,E1 15393.942,E2 15393.942} C_VEL
LIN {X 0,Y 319.95,Z 849.151,A -85,B 0,C 180,E1 15390.716,E2 15390.716} C_VEL
LIN {X 0,Y 319.947,Z 848.715,A -85,B 0,C 180,E1 15386.955,E2 15386.955} C_VEL
LIN {X 0,Y 319.962,Z 846.875,A -85,B 0,C 180,E1 15383.541,E2 15383.541} C_VEL
LIN {X 0,Y 320.117,Z 843.971,A -85,B 0,C 180,E1 15380.29,E2 15380.29} C_VEL
LIN {X 0,Y 320.535,Z 839.896,A -85,B 0,C 180,E1 15377.021,E2 15377.021} C_VEL
LIN {X 0,Y 321.564,Z 833.632,A -85,B 0,C 180,E1 15373.192,E2 15373.192} C_VEL
LIN {X 0,Y 323.238,Z 825.831,A -85,B 0,C 180,E1 15369.542,E2 15369.542} C_VEL
LIN {X 0,Y 325.305,Z 817.89,A -85,B 0,C 180,E1 15366.45,E2 15366.45} C_VEL
LIN {X 0,Y 328.581,Z 806.828,A -85,B 0,C 180,E1 15362.843,E2 15362.843} C_VEL
LIN {X 0,Y 332.345,Z 794.84,A -85,B 0,C 180,E1 15359.641,E2 15359.641} C_VEL
LIN {X 0,Y 336.126,Z 783.377,A -85,B 0,C 180,E1 15357.019,E2 15357.019} C_VEL
LIN {X 0,Y 341.274,Z 767.958,A -85,B 0,C 180,E1 15354.027,E2 15354.027} C_VEL
LIN {X 0,Y 346.148,Z 752.977,A -85,B 0,C 180,E1 15351.61,E2 15351.61} C_VEL
LIN {X 0,Y 350.6,Z 738.891,A -85,B 0,C 180,E1 15349.658,E2 15349.658} C_VEL
LIN {X 0,Y 356.12,Z 720.43,A -85,B 0,C 180,E1 15347.491,E2 15347.491} C_VEL
LIN {X 0,Y 360.828,Z 703.112,A -85,B 0,C 180,E1 15345.822,E2 15345.822} C_VEL
LIN {X 0,Y 364.978,Z 686.445,A -85,B 0,C 180,E1 15344.47,E2 15344.47} C_VEL
LIN {X 0,Y 369.385,Z 666.753,A -85,B 0,C 180,E1 15343.149,E2 15343.149} C_VEL
LIN {X 0,Y 373.139,Z 646.218,A -85,B 0,C 180,E1 15342.079,E2 15342.079} C_VEL
LIN {X 0,Y 375.856,Z 628.418,A -85,B 0,C 180,E1 15341.353,E2 15341.353} C_VEL
LIN {X 0,Y 378.431,Z 606.752,A -85,B 0,C 180,E1 15340.688,E2 15340.688} C_VEL
LIN {X 0,Y 380.575,Z 570.185,A -85,B 0,C 180,E1 15339.922,E2 15339.922} C_VEL
LIN {X 0,Y 389.671,Z 394.824,A -85,B 0,C 180,E1 15336.471,E2 15336.471} C_VEL
LIN {X 0,Y 380.665,Z 378.035,A -85,B 0,C 180,E1 15334.064,E2 15334.064} C_VEL
LIN {X 0,Y 372.536,Z 364.322,A -85,B 0,C 180,E1 15331.698,E2 15331.698} C_VEL
LIN {X 0,Y 366.041,Z 354.016,A -85,B 0,C 180,E1 15329.631,E2 15329.631} C_VEL
LIN {X 0,Y 358.635,Z 342.934,A -85,B 0,C 180,E1 15327.029,E2 15327.029} C_VEL
LIN {X 0,Y 354.139,Z 337.348,A -85,B 0,C 180,E1 15325.324,E2 15325.324} C_VEL
LIN {X 0,Y 350.47,Z 332.666,A -85,B 0,C 180,E1 15323.809,E2 15323.809} C_VEL
LIN {X 0,Y 346.366,Z 328.153,A -85,B 0,C 180,E1 15321.996,E2 15321.996} C_VEL
LIN {X 0,Y 345.008,Z 326.177,A -85,B 0,C 180,E1 15321.328,E2 15321.328} C_VEL
LIN {X 0,Y 341.674,Z 322.878,A -85,B 0,C 180,E1 15319.666,E2 15319.666} C_VEL
LIN {X 0,Y 340.002,Z 320.108,A -85,B 0,C 180,E1 15318.696,E2 15318.696} C_VEL
LIN {X 0,Y 336.741,Z 317.642,A -85,B 0,C 180,E1 15316.828,E2 15316.828} C_VEL
LIN {X 0,Y 334.288,Z 313.641,A -85,B 0,C 180,E1 15315.083,E2 15315.083} C_VEL
LIN {X 0,Y 330.717,Z 311.222,A -85,B 0,C 180,E1 15312.395,E2 15312.395} C_VEL
LIN {X 0,Y 329.024,Z 308.36,A -85,B 0,C 180,E1 15310.683,E2 15310.683} C_VEL
LIN {X 0,Y 327.944,Z 306.943,A -85,B 0,C 180,E1 15309.476,E2 15309.476} C_VEL
LIN {X 0,Y 323.705,Z 303.984,A -85,B 0,C 180,E1 15301.062,E2 15301.062} C_VEL
LIN {X 0,Y 324.014,Z 304.34,A -85,B 0,C 180,E1 15296.816,E2 15296.816} C_VEL
LIN {X 0,Y 328.339,Z 307.283,A -85,B 0,C 180,E1 15289.65,E2 15289.65} C_VEL
LIN {X 0,Y 329.329,Z 309.071,A -85,B 0,C 180,E1 15288.53,E2 15288.53} C_VEL
LIN {X 0,Y 331.426,Z 311.91,A -85,B 0,C 180,E1 15286.568,E2 15286.568} C_VEL
LIN {X 0,Y 334.712,Z 314.094,A -85,B 0,C 180,E1 15284.182,E2 15284.182} C_VEL
LIN {X 0,Y 336.884,Z 317.783,A -85,B 0,C 180,E1 15282.646,E2 15282.646} C_VEL
LIN {X 0,Y 340.101,Z 320.162,A -85,B 0,C 180,E1 15280.776,E2 15280.776} C_VEL
LIN {X 0,Y 341.106,Z 320.993,A -85,B 0,C 180,E1 15280.203,E2 15280.203} C_VEL
LIN {X 0,Y 343.655,Z 324.727,A -85,B 0,C 180,E1 15278.494,E2 15278.494} C_VEL
LIN {X 0,Y 346.837,Z 326.999,A -85,B 0,C 180,E1 15276.378,E2 15276.378} C_VEL
LIN {X 0,Y 348.298,Z 327.893,A -85,B 0,C 180,E1 15275.311,E2 15275.311} C_VEL
LIN {X 0,Y 350.413,Z 331.16,A -85,B 0,C 180,E1 15273.477,E2 15273.477} C_VEL
LIN {X 0,Y 352.885,Z 333.338,A -85,B 0,C 180,E1 15271.205,E2 15271.205} C_VEL
LIN {X 0,Y 355.704,Z 335.036,A -85,B 0,C 180,E1 15268.396,E2 15268.396} C_VEL
LIN {X 0,Y 357.646,Z 338.362,A -85,B 0,C 180,E1 15266.197,E2 15266.197} C_VEL
LIN {X 0,Y 360.51,Z 340.715,A -85,B 0,C 180,E1 15263.197,E2 15263.197} C_VEL
LIN {X 0,Y 362.634,Z 341.93,A -85,B 0,C 180,E1 15260.948,E2 15260.948} C_VEL
LIN {X 0,Y 364.838,Z 345.554,A -85,B 0,C 180,E1 15258.244,E2 15258.244} C_VEL
LIN {X 0,Y 367.647,Z 347.755,A -85,B 0,C 180,E1 15254.998,E2 15254.998} C_VEL
LIN {X 0,Y 369.717,Z 348.927,A -85,B 0,C 180,E1 15252.538,E2 15252.538} C_VEL
LIN {X 0,Y 371.457,Z 351.954,A -85,B 0,C 180,E1 15250.142,E2 15250.142} C_VEL
LIN {X 0,Y 373.777,Z 354.175,A -85,B 0,C 180,E1 15247.003,E2 15247.003} C_VEL
LIN {X 0,Y 376.424,Z 355.509,A -85,B 0,C 180,E1 15243.355,E2 15243.355} C_VEL
LIN {X 0,Y 377.428,Z 356.928,A -85,B 0,C 180,E1 15241.748,E2 15241.748} C_VEL
LIN {X 0,Y 379.269,Z 359.729,A -85,B 0,C 180,E1 15238.5,E2 15238.5} C_VEL
LIN {X 0,Y 381.167,Z 361.388,A -85,B 0,C 180,E1 15234.981,E2 15234.981} C_VEL
LIN {X 0,Y 383.058,Z 362.303,A -85,B 0,C 180,E1 15231.277,E2 15231.277} C_VEL
LIN {X 0,Y 384.352,Z 363.209,A -85,B 0,C 180,E1 15228.189,E2 15228.189} C_VEL
LIN {X 0,Y 385.505,Z 365.288,A -85,B 0,C 180,E1 15224.665,E2 15224.665} C_VEL
LIN {X 0,Y 386.412,Z 366.66,A -85,B 0,C 180,E1 15221.039,E2 15221.039} C_VEL
LIN {X 0,Y 387.099,Z 367.414,A -85,B 0,C 180,E1 15217.569,E2 15217.569} C_VEL
LIN {X 0,Y 387.554,Z 367.822,A -85,B 0,C 180,E1 15213.846,E2 15213.846} C_VEL
LIN {X 0,Y 387.721,Z 367.93,A -85,B 0,C 180,E1 15210.296,E2 15210.296} C_VEL
LIN {X 0,Y 387.597,Z 367.827,A -85,B 0,C 180,E1 15206.673,E2 15206.673} C_VEL
LIN {X 0,Y 387.209,Z 367.482,A -85,B 0,C 180,E1 15203.178,E2 15203.178} C_VEL
LIN {X 0,Y 386.542,Z 366.803,A -85,B 0,C 180,E1 15199.568,E2 15199.568} C_VEL
LIN {X 0,Y 385.668,Z 365.668,A -85,B 0,C 180,E1 15196.049,E2 15196.049} C_VEL
LIN {X 0,Y 384.562,Z 363.606,A -85,B 0,C 180,E1 15192.447,E2 15192.447} C_VEL
LIN {X 0,Y 383.44,Z 362.454,A -85,B 0,C 180,E1 15189.549,E2 15189.549} C_VEL
LIN {X 0,Y 381.679,Z 361.642,A -85,B 0,C 180,E1 15185.88,E2 15185.88} C_VEL
LIN {X 0,Y 379.751,Z 360.247,A -85,B 0,C 180,E1 15182.394,E2 15182.394} C_VEL
LIN {X 0,Y 377.991,Z 357.981,A -85,B 0,C 180,E1 15179.281,E2 15179.281} C_VEL
LIN {X 0,Y 376.655,Z 355.707,A -85,B 0,C 180,E1 15177.018,E2 15177.018} C_VEL
LIN {X 0,Y 373.923,Z 354.281,A -85,B 0,C 180,E1 15173.205,E2 15173.205} C_VEL
LIN {X 0,Y 371.548,Z 352.061,A -85,B 0,C 180,E1 15169.973,E2 15169.973} C_VEL
LIN {X 0,Y 369.888,Z 349.246,A -85,B 0,C 180,E1 15167.696,E2 15167.696} C_VEL
LIN {X 0,Y 368.751,Z 348.288,A -85,B 0,C 180,E1 15166.258,E2 15166.258} C_VEL
LIN {X 0,Y 365.994,Z 346.623,A -85,B 0,C 180,E1 15163.076,E2 15163.076} C_VEL
LIN {X 0,Y 363.839,Z 344.142,A -85,B 0,C 180,E1 15160.535,E2 15160.535} C_VEL
LIN {X 0,Y 362.244,Z 341.52,A -85,B 0,C 180,E1 15158.594,E2 15158.594} C_VEL
LIN {X 0,Y 359.08,Z 339.744,A -85,B 0,C 180,E1 15155.33,E2 15155.33} C_VEL
LIN {X 0,Y 356.747,Z 337.028,A -85,B 0,C 180,E1 15152.776,E2 15152.776} C_VEL
LIN {X 0,Y 355.318,Z 334.572,A -85,B 0,C 180,E1 15151.183,E2 15151.183} C_VEL
LIN {X 0,Y 351.806,Z 332.571,A -85,B 0,C 180,E1 15147.781,E2 15147.781} C_VEL
LIN {X 0,Y 350.661,Z 331.428,A -85,B 0,C 180,E1 15146.747,E2 15146.747} C_VEL
LIN {X 0,Y 349.584,Z 331.336,A -85,B 0,C 180,E1 15145.911,E2 15145.911} C_VEL
LIN {X 0,Y 345.756,Z 334.505,A -85,B 0,C 180,E1 15143.547,E2 15143.547} C_VEL
LIN {X 0,Y 344.787,Z 334.431,A -85,B 0,C 180,E1 15142.943,E2 15142.943} C_VEL
LIN {X 0,Y 341.572,Z 331.74,A -85,B 0,C 180,E1 15140.834,E2 15140.834} C_VEL
LIN {X 0,Y 338.878,Z 328.044,A -85,B 0,C 180,E1 15139.117,E2 15139.117} C_VEL
LIN {X 0,Y 335.525,Z 325.625,A -85,B 0,C 180,E1 15137.159,E2 15137.159} C_VEL
LIN {X 0,Y 333.093,Z 321.614,A -85,B 0,C 180,E1 15135.406,E2 15135.406} C_VEL
LIN {X 0,Y 329.185,Z 318.715,A -85,B 0,C 180,E1 15132.365,E2 15132.365} C_VEL
LIN {X 0,Y 327.216,Z 315.131,A -85,B 0,C 180,E1 15130.208,E2 15130.208} C_VEL
LIN {X 0,Y 322.761,Z 311.979,A -85,B 0,C 180,E1 15121.775,E2 15121.775} C_VEL
LIN {X 0,Y 322.932,Z 312.175,A -85,B 0,C 180,E1 15117.693,E2 15117.693} C_VEL
LIN {X 0,Y 327.286,Z 315.211,A -85,B 0,C 180,E1 15110.149,E2 15110.149} C_VEL
LIN {X 0,Y 329.456,Z 319.024,A -85,B 0,C 180,E1 15107.824,E2 15107.824} C_VEL
LIN {X 0,Y 333.185,Z 321.838,A -85,B 0,C 180,E1 15104.955,E2 15104.955} C_VEL
LIN {X 0,Y 335.638,Z 325.779,A -85,B 0,C 180,E1 15103.204,E2 15103.204} C_VEL
LIN {X 0,Y 338.581,Z 328.166,A -85,B 0,C 180,E1 15101.491,E2 15101.491} C_VEL
LIN {X 0,Y 341.607,Z 332.407,A -85,B 0,C 180,E1 15099.795,E2 15099.795} C_VEL
LIN {X 0,Y 343.779,Z 334.521,A -85,B 0,C 180,E1 15098.726,E2 15098.726} C_VEL
LIN {X 0,Y 347.174,Z 338.856,A -85,B 0,C 180,E1 15097.12,E2 15097.12} C_VEL
LIN {X 0,Y 348.674,Z 340.53,A -85,B 0,C 180,E1 15096.465,E2 15096.465} C_VEL
LIN {X 0,Y 353.553,Z 346.73,A -85,B 0,C 180,E1 15094.443,E2 15094.443} C_VEL
LIN {X 0,Y 357.735,Z 352.218,A -85,B 0,C 180,E1 15092.853,E2 15092.853} C_VEL
LIN {X 0,Y 365.873,Z 364.981,A -85,B 0,C 180,E1 15089.993,E2 15089.993} C_VEL
LIN {X 0,Y 373.644,Z 377.934,A -85,B 0,C 180,E1 15087.552,E2 15087.552} C_VEL
LIN {X 0,Y 382.347,Z 393.773,A -85,B 0,C 180,E1 15085.062,E2 15085.062} C_VEL
LIN {X 0,Y 384.759,Z 398.736,A -85,B 0,C 180,E1 15084.4,E2 15084.4} C_VEL
LIN {X 0,Y 373.694,Z 600.484,A -85,B 0,C 180,E1 15080.385,E2 15080.385} C_VEL
LIN {X 0,Y 371.321,Z 623.208,A -85,B 0,C 180,E1 15079.758,E2 15079.758} C_VEL
LIN {X 0,Y 368.315,Z 642.835,A -85,B 0,C 180,E1 15078.996,E2 15078.996} C_VEL
LIN {X 0,Y 365.143,Z 660.057,A -85,B 0,C 180,E1 15078.141,E2 15078.141} C_VEL
LIN {X 0,Y 360.812,Z 680.377,A -85,B 0,C 180,E1 15076.883,E2 15076.883} C_VEL
LIN {X 0,Y 355.736,Z 700.252,A -85,B 0,C 180,E1 15075.323,E2 15075.323} C_VEL
LIN {X 0,Y 351.156,Z 716.589,A -85,B 0,C 180,E1 15073.779,E2 15073.779} C_VEL
LIN {X 0,Y 345.599,Z 734.936,A -85,B 0,C 180,E1 15071.713,E2 15071.713} C_VEL
LIN {X 0,Y 340.091,Z 751.614,A -85,B 0,C 180,E1 15069.421,E2 15069.421} C_VEL
LIN {X 0,Y 335.456,Z 765.212,A -85,B 0,C 180,E1 15067.232,E2 15067.232} C_VEL
LIN {X 0,Y 330.071,Z 780.713,A -85,B 0,C 180,E1 15064.293,E2 15064.293} C_VEL
LIN {X 0,Y 325.621,Z 793.404,A -85,B 0,C 180,E1 15061.391,E2 15061.391} C_VEL
LIN {X 0,Y 321.942,Z 804.271,A -85,B 0,C 180,E1 15058.489,E2 15058.489} C_VEL
LIN {X 0,Y 318.194,Z 816.135,A -85,B 0,C 180,E1 15054.703,E2 15054.703} C_VEL
LIN {X 0,Y 315.752,Z 824.707,A -85,B 0,C 180,E1 15051.355,E2 15051.355} C_VEL
LIN {X 0,Y 314.094,Z 831.522,A -85,B 0,C 180,E1 15048.177,E2 15048.177} C_VEL
LIN {X 0,Y 312.797,Z 838.377,A -85,B 0,C 180,E1 15044.248,E2 15044.248} C_VEL
LIN {X 0,Y 312.166,Z 843.33,A -85,B 0,C 180,E1 15040.333,E2 15040.333} C_VEL
LIN {X 0,Y 311.991,Z 846.21,A -85,B 0,C 180,E1 15037.18,E2 15037.18} C_VEL
LIN {X 0,Y 311.947,Z 848.053,A -85,B 0,C 180,E1 15034.043,E2 15034.043} C_VEL
LIN {X 0,Y 311.954,Z 848.902,A -85,B 0,C 180,E1 15030.735,E2 15030.735} C_VEL
LIN {X 0,Y 311.949,Z 848.466,A -85,B 0,C 180,E1 15026.877,E2 15026.877} C_VEL
LIN {X 0,Y 311.966,Z 846.625,A -85,B 0,C 180,E1 15023.375,E2 15023.375} C_VEL
LIN {X 0,Y 312.136,Z 843.72,A -85,B 0,C 180,E1 15020.039,E2 15020.039} C_VEL
LIN {X 0,Y 312.596,Z 839.642,A -85,B 0,C 180,E1 15016.686,E2 15016.686} C_VEL
LIN {X 0,Y 313.715,Z 833.377,A -85,B 0,C 180,E1 15012.759,E2 15012.759} C_VEL
LIN {X 0,Y 315.52,Z 825.575,A -85,B 0,C 180,E1 15009.018,E2 15009.018} C_VEL
LIN {X 0,Y 317.733,Z 817.633,A -85,B 0,C 180,E1 15005.853,E2 15005.853} C_VEL
LIN {X 0,Y 321.221,Z 806.57,A -85,B 0,C 180,E1 15002.167,E2 15002.167} C_VEL
LIN {X 0,Y 325.215,Z 794.582,A -85,B 0,C 180,E1 14998.903,E2 14998.903} C_VEL
LIN {X 0,Y 329.198,Z 783.123,A -85,B 0,C 180,E1 14996.234,E2 14996.234} C_VEL
LIN {X 0,Y 334.588,Z 767.801,A -85,B 0,C 180,E1 14993.213,E2 14993.213} C_VEL
LIN {X 0,Y 339.722,Z 752.721,A -85,B 0,C 180,E1 14990.746,E2 14990.746} C_VEL
LIN {X 0,Y 344.573,Z 738.02,A -85,B 0,C 180,E1 14988.691,E2 14988.691} C_VEL
LIN {X 0,Y 350.599,Z 718.521,A -85,B 0,C 180,E1 14986.416,E2 14986.416} C_VEL
LIN {X 0,Y 355.262,Z 701.99,A -85,B 0,C 180,E1 14984.829,E2 14984.829} C_VEL
LIN {X 0,Y 359.585,Z 685.206,A -85,B 0,C 180,E1 14983.472,E2 14983.472} C_VEL
LIN {X 0,Y 364.51,Z 663.355,A -85,B 0,C 180,E1 14982.042,E2 14982.042} C_VEL
LIN {X 0,Y 367.829,Z 645.694,A -85,B 0,C 180,E1 14981.134,E2 14981.134} C_VEL
LIN {X 0,Y 370.608,Z 628.049,A -85,B 0,C 180,E1 14980.415,E2 14980.415} C_VEL
LIN {X 0,Y 373.26,Z 606.334,A -85,B 0,C 180,E1 14979.749,E2 14979.749} C_VEL
LIN {X 0,Y 375.521,Z 568.959,A -85,B 0,C 180,E1 14978.962,E2 14978.962} C_VEL
LIN {X 0,Y 384.699,Z 398.334,A -85,B 0,C 180,E1 14975.575,E2 14975.575} C_VEL
LIN {X 0,Y 376.29,Z 382.677,A -85,B 0,C 180,E1 14973.232,E2 14973.232} C_VEL
LIN {X 0,Y 369.364,Z 370.691,A -85,B 0,C 180,E1 14971.133,E2 14971.133} C_VEL
LIN {X 0,Y 363.117,Z 360.585,A -85,B 0,C 180,E1 14969.078,E2 14969.078} C_VEL
LIN {X 0,Y 356.161,Z 349.977,A -85,B 0,C 180,E1 14966.556,E2 14966.556} C_VEL
LIN {X 0,Y 351.654,Z 344.332,A -85,B 0,C 180,E1 14964.796,E2 14964.796} C_VEL
LIN {X 0,Y 347.532,Z 339.172,A -85,B 0,C 180,E1 14963.034,E2 14963.034} C_VEL
LIN {X 0,Y 344.009,Z 334.912,A -85,B 0,C 180,E1 14961.393,E2 14961.393} C_VEL
LIN {X 0,Y 342.896,Z 333.516,A -85,B 0,C 180,E1 14960.839,E2 14960.839} C_VEL
LIN {X 0,Y 339.529,Z 329.816,A -85,B 0,C 180,E1 14959.079,E2 14959.079} C_VEL
LIN {X 0,Y 338.159,Z 327.681,A -85,B 0,C 180,E1 14958.265,E2 14958.265} C_VEL
LIN {X 0,Y 335.004,Z 325.026,A -85,B 0,C 180,E1 14956.382,E2 14956.382} C_VEL
LIN {X 0,Y 332.845,Z 321.401,A -85,B 0,C 180,E1 14954.794,E2 14954.794} C_VEL
LIN {X 0,Y 329.362,Z 318.918,A -85,B 0,C 180,E1 14952.091,E2 14952.091} C_VEL
LIN {X 0,Y 327.58,Z 315.721,A -85,B 0,C 180,E1 14950.197,E2 14950.197} C_VEL
LIN {X 0,Y 326.217,Z 314.537,A -85,B 0,C 180,E1 14948.638,E2 14948.638} C_VEL
LIN {X 0,Y 322.713,Z 311.895,A -85,B 0,C 180,E1 14940.888,E2 14940.888} C_VEL
LIN {X 0,Y 323.092,Z 312.351,A -85,B 0,C 180,E1 14936.609,E2 14936.609} C_VEL
LIN {X 0,Y 327.212,Z 315.165,A -85,B 0,C 180,E1 14929.792,E2 14929.792} C_VEL
LIN {X 0,Y 329.657,Z 319.233,A -85,B 0,C 180,E1 14927.208,E2 14927.208} C_VEL
LIN {X 0,Y 333.196,Z 321.85,A -85,B 0,C 180,E1 14924.51,E2 14924.51} C_VEL
LIN {X 0,Y 335.654,Z 325.768,A -85,B 0,C 180,E1 14922.759,E2 14922.759} C_VEL
LIN {X 0,Y 339.496,Z 328.689,A -85,B 0,C 180,E1 14920.517,E2 14920.517} C_VEL
LIN {X 0,Y 342.276,Z 332.49,A -85,B 0,C 180,E1 14918.723,E2 14918.723} C_VEL
LIN {X 0,Y 345.672,Z 334.892,A -85,B 0,C 180,E1 14916.474,E2 14916.474} C_VEL
LIN {X 0,Y 346.905,Z 335.672,A -85,B 0,C 180,E1 14915.569,E2 14915.569} C_VEL
LIN {X 0,Y 349.192,Z 338.998,A -85,B 0,C 180,E1 14913.652,E2 14913.652} C_VEL
LIN {X 0,Y 351.799,Z 341.246,A -85,B 0,C 180,E1 14911.294,E2 14911.294} C_VEL
LIN {X 0,Y 354.478,Z 342.81,A -85,B 0,C 180,E1 14908.64,E2 14908.64} C_VEL
LIN {X 0,Y 356.443,Z 346.154,A -85,B 0,C 180,E1 14906.417,E2 14906.417} C_VEL
LIN {X 0,Y 359.499,Z 348.654,A -85,B 0,C 180,E1 14903.224,E2 14903.224} C_VEL
LIN {X 0,Y 361.508,Z 349.832,A -85,B 0,C 180,E1 14901.11,E2 14901.11} C_VEL
LIN {X 0,Y 363.791,Z 353.496,A -85,B 0,C 180,E1 14898.308,E2 14898.308} C_VEL
LIN {X 0,Y 366.607,Z 355.678,A -85,B 0,C 180,E1 14895.059,E2 14895.059} C_VEL
LIN {X 0,Y 368.612,Z 356.804,A -85,B 0,C 180,E1 14892.686,E2 14892.686} C_VEL
LIN {X 0,Y 370.271,Z 359.72,A -85,B 0,C 180,E1 14890.396,E2 14890.396} C_VEL
LIN {X 0,Y 372.545,Z 361.957,A -85,B 0,C 180,E1 14887.339,E2 14887.339} C_VEL
LIN {X 0,Y 375.194,Z 363.335,A -85,B 0,C 180,E1 14883.752,E2 14883.752} C_VEL
LIN {X 0,Y 376.148,Z 364.411,A -85,B 0,C 180,E1 14882.205,E2 14882.205} C_VEL
LIN {X 0,Y 377.909,Z 367.309,A -85,B 0,C 180,E1 14879.131,E2 14879.131} C_VEL
LIN {X 0,Y 379.878,Z 369.107,A -85,B 0,C 180,E1 14875.572,E2 14875.572} C_VEL
LIN {X 0,Y 381.76,Z 370.095,A -85,B 0,C 180,E1 14871.995,E2 14871.995} C_VEL
LIN {X 0,Y 383.259,Z 370.989,A -85,B 0,C 180,E1 14868.558,E2 14868.558} C_VEL
LIN {X 0,Y 384.371,Z 373.048,A -85,B 0,C 180,E1 14865.077,E2 14865.077} C_VEL
LIN {X 0,Y 385.342,Z 374.505,A -85,B 0,C 180,E1 14861.525,E2 14861.525} C_VEL
